FUNCTION "FC_LoadConfig" : Void
{ S7_Optimized_Access := 'TRUE' }
VERSION : 1.2
// =============================================================================
// Version_Recipe -- 00_Configuration.scl
// Central machine configuration -- called ONCE by OB100 (Startup) on every
// PLC power-up or program download.
//
// This file writes physical machine parameters (speed, limits, calibration, etc.)
// to DBs at PLC startup. Parameters that can be changed at runtime from HMI
// are NOT written here -- they remain as the DB initial values and revert to
// their initial values on warm-restart (NON_RETAIN DB).
//
// â”€â”€â”€ WHERE TO LOOK â”€â”€â”€â”€â”€â”€â”€â”€â”€â”€â”€â”€â”€â”€â”€â”€â”€â”€â”€â”€â”€â”€â”€â”€â”€â”€â”€â”€â”€â”€â”€â”€â”€â”€â”€â”€â”€â”€â”€â”€â”€â”€â”€â”€â”€â”€â”€â”€â”€â”€â”€â”€â”€â”€â”€â”€â”€â”€â”€
//   Maximum axis velocity        â†’ Section 1: MaxVelocity, RapidVelocity
//   Homing speed and mode        â†’ Section 2: HomeVelocity, HomingMode
//   Tool slot and angle settings â†’ Section 3: ToolCount, AutoCalcAngles
//   Spindle min/max RPM          â†’ Section 4: MinSpeed, MaxSpeed
//   Jog speed and step size      â†’ Section 5: JogSpeed, JogIncrement
//   Linear ruler stroke          â†’ Section 6: Phys_Max
//   Cylinder config reference    â†’ Section 7: see 02_DataBlocks.scl DB_Cylinder1
//   HMI initial values           â†’ Section 8: FeedrateOverride, ProductSelect
//   Test/commissioning bypass    â†’ Section 9: Bypass_EStop, Bypass_Door...
//   All timer PT values          â†’ Section 10: cylinder waits + process timeouts
//
// â”€â”€â”€ HMI SCREEN MAP â”€â”€â”€â”€â”€â”€â”€â”€â”€â”€â”€â”€â”€â”€â”€â”€â”€â”€â”€â”€â”€â”€â”€â”€â”€â”€â”€â”€â”€â”€â”€â”€â”€â”€â”€â”€â”€â”€â”€â”€â”€â”€â”€â”€â”€â”€â”€â”€â”€â”€â”€â”€â”€â”€â”€â”€â”€â”€
// Lists which tags are used on which HMI screen.
// "(â†’PLC)" = HMI writes, PLC reads  |  "(PLCâ†’)" = PLC writes, HMI reads (read-only)
//
// â”Œâ”€ MAIN SCREEN / STATUS LAMPS â”€â”€â”€â”€â”€â”€â”€â”€â”€â”€â”€â”€â”€â”€â”€â”€â”€â”€â”€â”€â”€â”€â”€â”€â”€â”€â”€â”€â”€â”€â”€â”€â”€â”€â”€â”€â”€â”€â”€â”€â”€â”€â”€â”€â”
// â”‚  DB_HMI.StatusMsg          (String[50])  PLCâ†’  "Running/Stopped/Errorâ€¦"â”‚
// â”‚  DB_HMI.IsRunning          (Bool)        PLCâ†’  Green lamp               â”‚
// â”‚  DB_HMI.IsPaused           (Bool)        PLCâ†’  Yellow lamp              â”‚
// â”‚  DB_HMI.HasError           (Bool)        PLCâ†’  Red lamp                 â”‚
// â”‚  DB_HMI.ActualX            (Real, mm)    PLCâ†’  X axis current position  â”‚
// â”‚  DB_HMI.ActualZ            (Real, mm)    PLCâ†’  Z axis current position  â”‚
// â”‚  DB_HMI.CurrentLine        (Int)         PLCâ†’  Active recipe line       â”‚
// â”‚  DB_HMI.ProgressPercent    (Real, %)     PLCâ†’  Progress bar             â”‚
// â”‚  DB_HMI.ElapsedSeconds     (DInt, s)     PLCâ†’  Cycle elapsed time       â”‚
// â”‚  DB_HMI.CycleCount         (Int)         PLCâ†’  Completed cycle count    â”‚
// â””â”€â”€â”€â”€â”€â”€â”€â”€â”€â”€â”€â”€â”€â”€â”€â”€â”€â”€â”€â”€â”€â”€â”€â”€â”€â”€â”€â”€â”€â”€â”€â”€â”€â”€â”€â”€â”€â”€â”€â”€â”€â”€â”€â”€â”€â”€â”€â”€â”€â”€â”€â”€â”€â”€â”€â”€â”€â”€â”€â”€â”€â”€â”€â”€â”€â”€â”€â”€â”€â”€â”€â”€â”€â”€â”˜
//
// â”Œâ”€ MAIN SCREEN / BUTTONS â”€â”€â”€â”€â”€â”€â”€â”€â”€â”€â”€â”€â”€â”€â”€â”€â”€â”€â”€â”€â”€â”€â”€â”€â”€â”€â”€â”€â”€â”€â”€â”€â”€â”€â”€â”€â”€â”€â”€â”€â”€â”€â”€â”€â”€â”€â”€â”€â”€â”€â”
// â”‚  DB_HMI.Btn_Start          (Bool)        â†’PLC  Start (rising edge)      â”‚
// â”‚  DB_HMI.Btn_Stop           (Bool)        â†’PLC  Stop (controlled stop)   â”‚
// â”‚  DB_HMI.Btn_Pause          (Bool)        â†’PLC  Pause                    â”‚
// â”‚  DB_HMI.Btn_Continue       (Bool)        â†’PLC  Resume from pause        â”‚
// â”‚  DB_HMI.Btn_AckError       (Bool)        â†’PLC  Acknowledge error + STOP â”‚
// â”‚  DB_HMI.Btn_Reset          (Bool)        â†’PLC  Full reset + STOPPED     â”‚
// â”‚  DB_HMI.ProductSelect      (Int, 1-5)    â†’PLC  Which program to run     â”‚
// â”‚  DB_HMI.FeedrateOverride   (Real, %)     â†’PLC  G1 speed multiplier      â”‚
// â”‚  DB_HMI.RapidOverride      (Real, %)     â†’PLC  G0 speed multiplier      â”‚
// â”‚  DB_HMI.SingleStepMode     (Bool)        â†’PLC  Line-by-line execution   â”‚
// â””â”€â”€â”€â”€â”€â”€â”€â”€â”€â”€â”€â”€â”€â”€â”€â”€â”€â”€â”€â”€â”€â”€â”€â”€â”€â”€â”€â”€â”€â”€â”€â”€â”€â”€â”€â”€â”€â”€â”€â”€â”€â”€â”€â”€â”€â”€â”€â”€â”€â”€â”€â”€â”€â”€â”€â”€â”€â”€â”€â”€â”€â”€â”€â”€â”€â”€â”€â”€â”€â”€â”€â”€â”€â”€â”˜
//
// â”Œâ”€ ERROR / ALARM SCREEN â”€â”€â”€â”€â”€â”€â”€â”€â”€â”€â”€â”€â”€â”€â”€â”€â”€â”€â”€â”€â”€â”€â”€â”€â”€â”€â”€â”€â”€â”€â”€â”€â”€â”€â”€â”€â”€â”€â”€â”€â”€â”€â”€â”€â”€â”€â”€â”€â”€â”€â”€â”
// â”‚  DB_Error.Active           (Bool)        PLCâ†’  Is there an active error? â”‚
// â”‚  DB_Error.Code             (Word, hex)   PLCâ†’  Error code (e.g. 0x0401) â”‚
// â”‚  DB_Error.Details          (String[80])  PLCâ†’  Error description text   â”‚
// â”‚  DB_Error.Severity         (Byte)        PLCâ†’  3=fatal, 2=error, 1=warn â”‚
// â”‚  DB_Error.Source           (String[20])  PLCâ†’  "Safety"/"Axis"/"Limit"  â”‚
// â”‚  DB_Error.TimeStamp        (DTL)         PLCâ†’  Error timestamp          â”‚
// â”‚  -- Alarm History (last 10) â”€â”€â”€â”€â”€â”€â”€â”€â”€â”€â”€â”€â”€â”€â”€â”€â”€â”€â”€â”€â”€â”€â”€â”€â”€â”€â”€â”€â”€â”€â”€â”€â”€â”€â”€â”€â”€â”€â”€â”€â”€â”€â”€â”€â”‚
// â”‚  DB_Error.History_Code[1..10]   (Word)   PLCâ†’  Last 10 error codes      â”‚
// â”‚  DB_Error.History_Details[1..10](String) PLCâ†’  Last 10 error details    â”‚
// â”‚  DB_Error.History_Time[1..10]   (DTL)    PLCâ†’  Last 10 error timestamps â”‚
// â””â”€â”€â”€â”€â”€â”€â”€â”€â”€â”€â”€â”€â”€â”€â”€â”€â”€â”€â”€â”€â”€â”€â”€â”€â”€â”€â”€â”€â”€â”€â”€â”€â”€â”€â”€â”€â”€â”€â”€â”€â”€â”€â”€â”€â”€â”€â”€â”€â”€â”€â”€â”€â”€â”€â”€â”€â”€â”€â”€â”€â”€â”€â”€â”€â”€â”€â”€â”€â”€â”€â”€â”€â”€â”€â”˜
//
// â”Œâ”€ MANUAL SCREEN / MOTION â”€â”€â”€â”€â”€â”€â”€â”€â”€â”€â”€â”€â”€â”€â”€â”€â”€â”€â”€â”€â”€â”€â”€â”€â”€â”€â”€â”€â”€â”€â”€â”€â”€â”€â”€â”€â”€â”€â”€â”€â”€â”€â”€â”€â”€â”€â”€â”€â”€â”
// â”‚  DB_Manual.ManualModeActive (Bool)       â†’PLC  Enable/disable manual modeâ”‚
// â”‚  DB_Manual.SelectedAxis    (Int, 0-3)    â†’PLC  0=X 1=Z 2=Tool 3=Spindle â”‚
// â”‚  DB_Manual.Btn_JogPlus     (Bool)        â†’PLC  Positive direction jog   â”‚
// â”‚  DB_Manual.Btn_JogMinus    (Bool)        â†’PLC  Negative direction jog   â”‚
// â”‚  DB_Manual.JogSpeed        (Real, mm/s)  â†’PLC  Jog speed                â”‚
// â”‚  DB_Manual.Btn_StepPlus    (Bool)        â†’PLC  +JogIncrement step       â”‚
// â”‚  DB_Manual.Btn_StepMinus   (Bool)        â†’PLC  -JogIncrement step       â”‚
// â”‚  DB_Manual.JogIncrement    (Real, mm)    â†’PLC  Step size                â”‚
// â”‚  DB_Manual.MoveToPosition  (Real, mm)    â†’PLC  Target absolute position â”‚
// â”‚  DB_Manual.Btn_MoveAbsolute(Bool)        â†’PLC  Start absolute move      â”‚
// â”‚  DB_Manual.Btn_HomeAll     (Bool)        â†’PLC  Home all axes             â”‚
// â”‚  DB_Manual.Btn_GoSafe      (Bool)        â†’PLC  Move to safe position    â”‚
// â”‚  DB_Manual.Btn_GoZero      (Bool)        â†’PLC  Move to zero position    â”‚
// â”‚  DB_Manual.SelectedAxisPos (Real, mm)    PLCâ†’  Selected axis position   â”‚
// â”‚  DB_Manual.SelectedAxisName(String)      PLCâ†’  "X" / "Z" / "Tool"      â”‚
// â”‚  DB_Manual.JogBusy         (Bool)        PLCâ†’  Motion in progress       â”‚
// â””â”€â”€â”€â”€â”€â”€â”€â”€â”€â”€â”€â”€â”€â”€â”€â”€â”€â”€â”€â”€â”€â”€â”€â”€â”€â”€â”€â”€â”€â”€â”€â”€â”€â”€â”€â”€â”€â”€â”€â”€â”€â”€â”€â”€â”€â”€â”€â”€â”€â”€â”€â”€â”€â”€â”€â”€â”€â”€â”€â”€â”€â”€â”€â”€â”€â”€â”€â”€â”€â”€â”€â”€â”€â”€â”˜
//
// â”Œâ”€ MANUAL SCREEN / SPINDLE â”€â”€â”€â”€â”€â”€â”€â”€â”€â”€â”€â”€â”€â”€â”€â”€â”€â”€â”€â”€â”€â”€â”€â”€â”€â”€â”€â”€â”€â”€â”€â”€â”€â”€â”€â”€â”€â”€â”€â”€â”€â”€â”€â”€â”€â”€â”€â”€â”
// â”‚  DB_Manual.Btn_SpindleStart(Bool)        â†’PLC  Start spindle            â”‚
// â”‚  DB_Manual.Btn_SpindleStop (Bool)        â†’PLC  Stop spindle             â”‚
// â”‚  DB_Manual.Manual_SpindleSpeed (Real,RPM)â†’PLC  Manual spindle speed     â”‚
// â”‚  DB_Manual.Manual_SpindleDir   (Int)     â†’PLC  1=CW, -1=CCW            â”‚
// â”‚  DB_Spindle.IsRunning      (Bool)        PLCâ†’  Spindle running          â”‚
// â”‚  DB_Spindle.AtSpeed        (Bool)        PLCâ†’  Speed stable             â”‚
// â”‚  DB_Spindle.ActualSpeed    (Real, RPM)   PLCâ†’  Current spindle speed    â”‚
// â””â”€â”€â”€â”€â”€â”€â”€â”€â”€â”€â”€â”€â”€â”€â”€â”€â”€â”€â”€â”€â”€â”€â”€â”€â”€â”€â”€â”€â”€â”€â”€â”€â”€â”€â”€â”€â”€â”€â”€â”€â”€â”€â”€â”€â”€â”€â”€â”€â”€â”€â”€â”€â”€â”€â”€â”€â”€â”€â”€â”€â”€â”€â”€â”€â”€â”€â”€â”€â”€â”€â”€â”€â”€â”€â”˜
//
// â”Œâ”€ MANUAL SCREEN / MANAGE (Drive Management) â”€â”€â”€â”€â”€â”€â”€â”€â”€â”€â”€â”€â”€â”€â”€â”€â”€â”€â”€â”€â”€â”€â”€â”€â”€â”€â”€â”€â”€â”
// â”‚  DB_HMI.Btn_Contactor_X    (Bool)        â†’PLC  X drive contactor        â”‚
// â”‚  DB_HMI.Btn_Contactor_Z    (Bool)        â†’PLC  Z drive contactor        â”‚
// â”‚  DB_HMI.Btn_Contactor_Tool (Bool)        â†’PLC  Tool drive contactor     â”‚
// â”‚  DB_HMI.Btn_Enable_X       (Bool)        â†’PLC  X drive enable signal    â”‚
// â”‚  DB_HMI.Btn_Enable_Z       (Bool)        â†’PLC  Z drive enable signal    â”‚
// â”‚  DB_HMI.Contactor_X_On     (Bool)        PLCâ†’  X contactor feedback     â”‚
// â”‚  DB_HMI.Contactor_Z_On     (Bool)        PLCâ†’  Z contactor feedback     â”‚
// â”‚  DB_HMI.Enable_X_On        (Bool)        PLCâ†’  X enable feedback        â”‚
// â”‚  NOTE: Contactor and Enable must be toggle buttons (maintained),         â”‚
// â”‚        NOT momentary.                                                    â”‚
// â””â”€â”€â”€â”€â”€â”€â”€â”€â”€â”€â”€â”€â”€â”€â”€â”€â”€â”€â”€â”€â”€â”€â”€â”€â”€â”€â”€â”€â”€â”€â”€â”€â”€â”€â”€â”€â”€â”€â”€â”€â”€â”€â”€â”€â”€â”€â”€â”€â”€â”€â”€â”€â”€â”€â”€â”€â”€â”€â”€â”€â”€â”€â”€â”€â”€â”€â”€â”€â”€â”€â”€â”€â”€â”€â”˜
//
// â”Œâ”€ TOOL PAGE â”€â”€â”€â”€â”€â”€â”€â”€â”€â”€â”€â”€â”€â”€â”€â”€â”€â”€â”€â”€â”€â”€â”€â”€â”€â”€â”€â”€â”€â”€â”€â”€â”€â”€â”€â”€â”€â”€â”€â”€â”€â”€â”€â”€â”€â”€â”€â”€â”€â”€â”€â”€â”€â”€â”€â”€â”€â”€â”€â”€â”€â”€â”
// â”‚  DB_MachineConfig.ToolCount         (Int, 1-4)  â†’PLC  Slot count        â”‚
// â”‚  DB_ToolConfig.AutoCalcAngles       (Bool)       â†’PLC  Auto angle calc  â”‚
// â”‚  DB_ToolConfig.ToolStepAngle_Calc   (Real, Â°)   PLCâ†’  Calculated step   â”‚
// â”‚  DB_ToolConfig.Tool1_Position       (Real, Â°)   PLCâ†’  Slot 1 angle      â”‚
// â”‚  DB_ToolConfig.Tool2_Position       (Real, Â°)   PLCâ†’  Slot 2 angle      â”‚
// â”‚  DB_ToolConfig.Tool3_Position       (Real, Â°)   PLCâ†’  Slot 3 angle      â”‚
// â”‚  DB_ToolConfig.Tool4_Position       (Real, Â°)   PLCâ†’  Slot 4 angle      â”‚
// â”‚  DB_HMI.ToolSlotCode[1..4]          (Int)        â†’PLC  Slot code input  â”‚
// â”‚  DB_HMI.Btn_ApplyToolConfig         (Bool)       â†’PLC  Apply code       â”‚
// â”‚  DB_ToolConfig.ToolCode_List[1..4]  (Int)        PLCâ†’  Active slot code â”‚
// â”‚  NOTE: While AutoCalcAngles=TRUE, tool angles cannot be changed from     â”‚
// â”‚        HMI -- they are overwritten every scan. Set FALSE for manual anglesâ”‚
// â””â”€â”€â”€â”€â”€â”€â”€â”€â”€â”€â”€â”€â”€â”€â”€â”€â”€â”€â”€â”€â”€â”€â”€â”€â”€â”€â”€â”€â”€â”€â”€â”€â”€â”€â”€â”€â”€â”€â”€â”€â”€â”€â”€â”€â”€â”€â”€â”€â”€â”€â”€â”€â”€â”€â”€â”€â”€â”€â”€â”€â”€â”€â”€â”€â”€â”€â”€â”€â”€â”€â”€â”€â”€â”€â”˜
//
// â”Œâ”€ CYLINDER PAGE â”€â”€â”€â”€â”€â”€â”€â”€â”€â”€â”€â”€â”€â”€â”€â”€â”€â”€â”€â”€â”€â”€â”€â”€â”€â”€â”€â”€â”€â”€â”€â”€â”€â”€â”€â”€â”€â”€â”€â”€â”€â”€â”€â”€â”€â”€â”€â”€â”€â”€â”€â”€â”€â”€â”€â”€â”€â”€â”
// â”‚  DB_Cylinder1.ValveType    (Byte)        â†’PLC  1=5/2  2=5/3_blocked     â”‚
// â”‚  DB_Cylinder1.Cmd_Extend   (Bool)        â†’PLC  Extend: move to setpoint â”‚
// â”‚  DB_Cylinder1.Cmd_ExtendFull(Bool)       â†’PLC  Extend: full stroke      â”‚
// â”‚  DB_Cylinder1.Cmd_Retract  (Bool)        â†’PLC  Retract                  â”‚
// â”‚  DB_Cylinder1.Timeout_Extend(Time)       â†’PLC  Extend timeout (T#5S)    â”‚
// â”‚  DB_Cylinder1.Timeout_Retract(Time)      â†’PLC  Retract timeout (T#5S)   â”‚
// â”‚  DB_Cylinder1.State        (Int)         PLCâ†’  -1=EStop 0=Idle          â”‚
// â”‚                                                  1=Extending 2=Retractingâ”‚
// â”‚                                                  3=AtSetpoint 4=AtRetractâ”‚
// â”‚                                                 10=ERROR                 â”‚
// â”‚  DB_Cylinder1.StateText    (String[14])  PLCâ†’  State text               â”‚
// â”‚  DB_Cylinder1.AtSetpoint   (Bool)        PLCâ†’  Locked at setpoint       â”‚
// â”‚  DB_Cylinder1.AtRetract    (Bool)        PLCâ†’  At retract end           â”‚
// â”‚  DB_Cylinder1.Error        (Bool)        PLCâ†’  Active error             â”‚
// â”‚  DB_Cylinder1.ErrorID      (Word)        PLCâ†’  0x0501/0502/0503         â”‚
// â”‚  DB_LinearRuler1.Value      (Real, mm)    PLCâ†’  Ruler position           â”‚
// â”‚  DB_LinearRuler1.Valid       (Bool)        PLCâ†’  Sensor healthy?         â”‚
// â”‚  NOTE: Cmd_Extend AND Cmd_Retract TRUE simultaneously â†’ Hold (conflict  â”‚
// â”‚        protection). Purchase BLOCKED CENTER valve -- cylinder is          â”‚
// â”‚        mechanically locked in hold. Do NOT use EXHAUST CENTER.          â”‚
// â””â”€â”€â”€â”€â”€â”€â”€â”€â”€â”€â”€â”€â”€â”€â”€â”€â”€â”€â”€â”€â”€â”€â”€â”€â”€â”€â”€â”€â”€â”€â”€â”€â”€â”€â”€â”€â”€â”€â”€â”€â”€â”€â”€â”€â”€â”€â”€â”€â”€â”€â”€â”€â”€â”€â”€â”€â”€â”€â”€â”€â”€â”€â”€â”€â”€â”€â”€â”€â”€â”€â”€â”€â”€â”€â”˜
//
// â”Œâ”€ RULER CALIBRATION (Setup Screen) â”€â”€â”€â”€â”€â”€â”€â”€â”€â”€â”€â”€â”€â”€â”€â”€â”€â”€â”€â”€â”€â”€â”€â”€â”€â”€â”€â”€â”€â”€â”€â”€â”€â”€â”€â”€â”€â”€â”
// â”‚  DB_LinearRuler1.Raw_Min      (Int)       â†’PLC  AI raw min value         â”‚
// â”‚  DB_LinearRuler1.Raw_Max      (Int)       â†’PLC  AI raw max value         â”‚
// â”‚  DB_LinearRuler1.Phys_Min     (Real, mm)  â†’PLC  Physical ref at Raw_Min  â”‚
// â”‚  DB_LinearRuler1.Phys_Max     (Real, mm)  â†’PLC  Physical ref at Raw_Max  â”‚
// â”‚  DB_LinearRuler1.InvertSignal (Bool)      â†’PLC  TRUE=0Vâ†’high physical    â”‚
// â”‚  DB_LinearRuler1.Value        (Real, mm)  PLCâ†’  Scaled position (mm)     â”‚
// â”‚  DB_LinearRuler1.Valid        (Bool)      PLCâ†’  Sensor within range?     â”‚
// â”‚  NOTE: S7-1200 standard AI: 0V=0, 10V=27648 (4-20mA: 4mA=5530,20mA=27648â”‚
// â””â”€â”€â”€â”€â”€â”€â”€â”€â”€â”€â”€â”€â”€â”€â”€â”€â”€â”€â”€â”€â”€â”€â”€â”€â”€â”€â”€â”€â”€â”€â”€â”€â”€â”€â”€â”€â”€â”€â”€â”€â”€â”€â”€â”€â”€â”€â”€â”€â”€â”€â”€â”€â”€â”€â”€â”€â”€â”€â”€â”€â”€â”€â”€â”€â”€â”€â”€â”€â”€â”€â”€â”€â”€â”€â”˜
//
// â”Œâ”€ MACHINE LIMITS (Setup Screen) â”€â”€â”€â”€â”€â”€â”€â”€â”€â”€â”€â”€â”€â”€â”€â”€â”€â”€â”€â”€â”€â”€â”€â”€â”€â”€â”€â”€â”€â”€â”€â”€â”€â”€â”€â”€â”€â”€â”€â”€â”€â”
// â”‚  DB_MachineConfig.SoftLimit_MinX  (Real, mm)  â†’PLC  X software min      â”‚
// â”‚  DB_MachineConfig.SoftLimit_MaxX  (Real, mm)  â†’PLC  X software max      â”‚
// â”‚  DB_MachineConfig.SoftLimit_MinZ  (Real, mm)  â†’PLC  Z software min      â”‚
// â”‚  DB_MachineConfig.SoftLimit_MaxZ  (Real, mm)  â†’PLC  Z software max      â”‚
// â”‚  DB_MachineConfig.HomeVelocity    (Real, mm/s)â†’PLC  Homing speed        â”‚
// â”‚  DB_MachineConfig.SafePos_X/Z     (Real, mm)  â†’PLC  "Go Safe" target    â”‚
// â”‚  NOTE: These values are not written by FC_LoadConfig. Use DB initial     â”‚
// â”‚        values or change from HMI. Reverts to DB initial on PLC restart. â”‚
// â””â”€â”€â”€â”€â”€â”€â”€â”€â”€â”€â”€â”€â”€â”€â”€â”€â”€â”€â”€â”€â”€â”€â”€â”€â”€â”€â”€â”€â”€â”€â”€â”€â”€â”€â”€â”€â”€â”€â”€â”€â”€â”€â”€â”€â”€â”€â”€â”€â”€â”€â”€â”€â”€â”€â”€â”€â”€â”€â”€â”€â”€â”€â”€â”€â”€â”€â”€â”€â”€â”€â”€â”€â”€â”€â”˜
//
// â”Œâ”€ PRODUCTION COUNTERS â”€â”€â”€â”€â”€â”€â”€â”€â”€â”€â”€â”€â”€â”€â”€â”€â”€â”€â”€â”€â”€â”€â”€â”€â”€â”€â”€â”€â”€â”€â”€â”€â”€â”€â”€â”€â”€â”€â”€â”€â”€â”€â”€â”€â”€â”€â”€â”€â”€â”€â”€â”€â”
// â”‚  DB_Production.TotalOK     (DInt)        PLCâ†’  Successful cycle count   â”‚
// â”‚  DB_Production.TotalNOK    (DInt)        PLCâ†’  Failed cycle count       â”‚
// â”‚  DB_Production.TotalStopped(DInt)        PLCâ†’  Operator stop count      â”‚
// â”‚  DB_Production.LastResult  (Byte)        PLCâ†’  1=OK, 2=NOK, 3=STOP      â”‚
// â”‚  DB_Production.LastErrorCode(Word)       PLCâ†’  Last error code          â”‚
// â”‚  DB_HMI.Btn_ProdReset      (Bool)        â†’PLC  Reset counters           â”‚
// â””â”€â”€â”€â”€â”€â”€â”€â”€â”€â”€â”€â”€â”€â”€â”€â”€â”€â”€â”€â”€â”€â”€â”€â”€â”€â”€â”€â”€â”€â”€â”€â”€â”€â”€â”€â”€â”€â”€â”€â”€â”€â”€â”€â”€â”€â”€â”€â”€â”€â”€â”€â”€â”€â”€â”€â”€â”€â”€â”€â”€â”€â”€â”€â”€â”€â”€â”€â”€â”€â”€â”€â”€â”€â”€â”˜
//
// â”Œâ”€ BYPASS / TEST MODE â”€â”€â”€â”€â”€â”€â”€â”€â”€â”€â”€â”€â”€â”€â”€â”€â”€â”€â”€â”€â”€â”€â”€â”€â”€â”€â”€â”€â”€â”€â”€â”€â”€â”€â”€â”€â”€â”€â”€â”€â”€â”€â”€â”€â”€â”€â”€â”€â”€â”€â”€â”€â”€â”
// â”‚  DB_HMI.Bypass_EStop       (Bool)        â†’PLC  âš ï¸ TEST ONLY             â”‚
// â”‚  DB_HMI.Bypass_Door        (Bool)        â†’PLC  âš ï¸ TEST ONLY             â”‚
// â”‚  DB_HMI.Bypass_AirPressure (Bool)        â†’PLC  âš ï¸ TEST ONLY             â”‚
// â”‚  DB_HMI.Bypass_Drives      (Bool)        â†’PLC  âš ï¸ TEST ONLY             â”‚
// â”‚  âš ï¸ The PLC does NOT clear bypasses while active. The operator must      â”‚
// â”‚     turn them off manually. Verify before going into production.         â”‚
// â”‚  NOTE: DB_HMI.Bypass_Spindle and Bypass_ToolChanger are defined but     â”‚
// â”‚        not used in the safety monitor -- do not connect them.            â”‚
// â””â”€â”€â”€â”€â”€â”€â”€â”€â”€â”€â”€â”€â”€â”€â”€â”€â”€â”€â”€â”€â”€â”€â”€â”€â”€â”€â”€â”€â”€â”€â”€â”€â”€â”€â”€â”€â”€â”€â”€â”€â”€â”€â”€â”€â”€â”€â”€â”€â”€â”€â”€â”€â”€â”€â”€â”€â”€â”€â”€â”€â”€â”€â”€â”€â”€â”€â”€â”€â”€â”€â”€â”€â”€â”€â”˜
// =============================================================================
// -----------------------------------------------------------------------------
// FC_LoadConfig -- Runs once at PLC startup (called by OB100)
// Values here can be thought of as the PLC "factory defaults".
// Parameters that can be changed at runtime from HMI are NOT written here --
// the initial value in the DB definition applies.
// -----------------------------------------------------------------------------

BEGIN


	// =========================================================================
	// SECTION 1 -- AXIS VELOCITY LIMITS (mm/s)
	// â”€â”€â”€â”€â”€â”€â”€â”€â”€â”€â”€â”€â”€â”€â”€â”€â”€â”€â”€â”€â”€â”€â”€â”€â”€â”€â”€â”€â”€â”€â”€â”€â”€â”€â”€â”€â”€â”€â”€â”€â”€â”€â”€â”€â”€â”€â”€â”€â”€â”€â”€â”€â”€â”€â”€â”€â”€â”€â”€â”€â”€â”€â”€â”€â”€â”€â”€â”€â”€â”€â”€â”€â”€
	// âš ï¸ These values MUST match the Technology Object (TO) settings in TIA Portal.
	//    If the TO has a different limit, the PLC may report an error.
	//    Should not be changed from HMI -- edit here instead.
	// â”€â”€â”€â”€â”€â”€â”€â”€â”€â”€â”€â”€â”€â”€â”€â”€â”€â”€â”€â”€â”€â”€â”€â”€â”€â”€â”€â”€â”€â”€â”€â”€â”€â”€â”€â”€â”€â”€â”€â”€â”€â”€â”€â”€â”€â”€â”€â”€â”€â”€â”€â”€â”€â”€â”€â”€â”€â”€â”€â”€â”€â”€â”€â”€â”€â”€â”€â”€â”€â”€â”€â”€â”€
	//  MaxVelocity   : Must match "Maximum velocity" in TO
	//  RapidVelocity : Used for G0 command (in recipe)
	//  MinVelocity   : Must match "Minimum velocity" in TO
	// =========================================================================
	"DB_MachineConfig".MaxVelocity := 40.0;   // mm/s -- match TO max velocity
	"DB_MachineConfig".RapidVelocity := 30.0;   // mm/s -- G0 (rapid move) speed
	"DB_MachineConfig".MinVelocity := 0.001;    // mm/s -- match TO min velocity
	"DB_MachineConfig".FeedrateConvFactor := 60.0;    // divisor: recipe F (mm/min) / this = axis velocity (mm/s)
	// Standard mm/minâ†’mm/s = divide by 60; adjust if TO uses different units

	// =========================================================================
	// SECTION 2 -- HOMING (REFERENCE SEEK)
	// â”€â”€â”€â”€â”€â”€â”€â”€â”€â”€â”€â”€â”€â”€â”€â”€â”€â”€â”€â”€â”€â”€â”€â”€â”€â”€â”€â”€â”€â”€â”€â”€â”€â”€â”€â”€â”€â”€â”€â”€â”€â”€â”€â”€â”€â”€â”€â”€â”€â”€â”€â”€â”€â”€â”€â”€â”€â”€â”€â”€â”€â”€â”€â”€â”€â”€â”€â”€â”€â”€â”€â”€â”€
	//  HomingMode:
	//    0 = Passive  â†’ Motor does not move, encoder is zeroed at current position
	//    2 = Active   â†’ Moves to reference switch, encoder is zeroed
	//    3 = Active+Zero â†’ Moves to reference switch, set to HomeOffset_X/Z value
	//                    (recommended mode for production)
	//
	//  HomeVelocity and HomeOffset_X/Z are defined as initial values in
	//  DB_MachineConfig and can be edited from the HMI Machine Limits screen.
	//  Writing here will always reset to the same value on restart.
	// =========================================================================
	"DB_Manual".HomingMode := 3;   // 0=Passive | 2=Active | 3=Active+Zero (recommended)
	"DB_MachineConfig".PostHome_Clearance := 0.0;  // mm -- clearance distance from PNP zone after homing
	"DB_MachineConfig".HomeVelocity := 5.0;         // mm/s -- speed for pre/post-homing clearance move
	// NOTE: MC_Home search speed comes from TO, PLC cannot change it
	"DB_MachineConfig".AlwaysHomeOnAutoStart := TRUE; // Home all axes on every auto start (set FALSE for fast test cycles)

	// =========================================================================
	// SECTION 3 -- TOOL CHANGER
	// â”€â”€â”€â”€â”€â”€â”€â”€â”€â”€â”€â”€â”€â”€â”€â”€â”€â”€â”€â”€â”€â”€â”€â”€â”€â”€â”€â”€â”€â”€â”€â”€â”€â”€â”€â”€â”€â”€â”€â”€â”€â”€â”€â”€â”€â”€â”€â”€â”€â”€â”€â”€â”€â”€â”€â”€â”€â”€â”€â”€â”€â”€â”€â”€â”€â”€â”€â”€â”€â”€â”€â”€â”€
	//  ToolCount: How many slots are physically installed (1-4)
	//    â†’ FC_ToolAngleCalc automatically calculates angles based on this value
	//    â†’ Can also be changed on the HMI Tool page (runtime)
	//
	//  AutoCalcAngles = TRUE  â†’ Equally spaced angles based on ToolCount
	//                           (2 slots: 0Â°/180Â°, 3 slots: 0Â°/120Â°/240Â°, etc.)
	//  AutoCalcAngles = FALSE â†’ Tool1..4_Position can be entered manually from HMI
	//                           (use when unequal angles are needed)
	//
	//  CurrentTool: Which slot is active at startup (usually 1)
	// =========================================================================
	"DB_MachineConfig".ToolCount := 3;     // Physical slot count
	"DB_ToolConfig".AutoCalcAngles := TRUE;  // Automatic angle calculation
	"DB_ToolConfig".CurrentTool := 1;     // Initial active slot

	// =========================================================================
	// SECTION 4 -- SPINDLE SPEED
	// â”€â”€â”€â”€â”€â”€â”€â”€â”€â”€â”€â”€â”€â”€â”€â”€â”€â”€â”€â”€â”€â”€â”€â”€â”€â”€â”€â”€â”€â”€â”€â”€â”€â”€â”€â”€â”€â”€â”€â”€â”€â”€â”€â”€â”€â”€â”€â”€â”€â”€â”€â”€â”€â”€â”€â”€â”€â”€â”€â”€â”€â”€â”€â”€â”€â”€â”€â”€â”€â”€â”€â”€â”€
	//  MinSpeed      : Commands below this value are clamped to this value
	//  MaxSpeed      : Commands above this value are clamped to this value
	//  DefaultSpeed  : Default speed in manual mode (initial Manual_SpindleSpeed)
	//  SpeedTolerance: Tolerance for "AtSpeed" decision -- keep small (Â±5% recommended)
	//  SpeedOverride : 100% = normal, can be changed at runtime from HMI
	//
	//  âš ï¸ MaxSpeed must not exceed motor or coupling component ratings
	// =========================================================================
	"DB_Spindle".MinSpeed := 100.0;   // RPM -- lower limit
	"DB_Spindle".MaxSpeed := 3000.0;  // RPM -- upper limit (do not exceed motor max)
	"DB_Spindle".DefaultSpeed := 1000.0;  // RPM -- manual mode initial value
	"DB_Spindle".SpeedTolerance := 5.0;     // % -- AtSpeed tolerance
	"DB_Spindle".SpeedOverride := 100.0;   // % -- 100% at startup (normal)
	"DB_MachineConfig".SpindleMaxRPM := 2400.0;  // RPM -- denominator for proportional MandrelLock wait (ITEM-28)
	"DB_MachineConfig".SpindleStopSafeTime := T#10S;   // Full-speed decel safety margin -- tune to measured VFD ramp + margin

	// =========================================================================
	// SECTION 5 -- MANUAL MODE DEFAULTS
	// â”€â”€â”€â”€â”€â”€â”€â”€â”€â”€â”€â”€â”€â”€â”€â”€â”€â”€â”€â”€â”€â”€â”€â”€â”€â”€â”€â”€â”€â”€â”€â”€â”€â”€â”€â”€â”€â”€â”€â”€â”€â”€â”€â”€â”€â”€â”€â”€â”€â”€â”€â”€â”€â”€â”€â”€â”€â”€â”€â”€â”€â”€â”€â”€â”€â”€â”€â”€â”€â”€â”€â”€â”€
	//  JogSpeed      : Speed used when jog button is pressed
	//                  Can be connected to a slider/input field on HMI Manual screen
	//  JogIncrement  : Distance traveled per press on "Step" button
	//  ToolStepAngle : Rotation angle for CW/CCW buttons on Manual Tool screen
	//                  (e.g. 90Â° can be used to step slot-to-slot)
	//  Manual_SpindleSpeed: Initial speed on manual spindle screen
	//  Manual_SpindleDir  : 1=CW (clockwise), -1=CCW (counter-clockwise)
	// =========================================================================
	"DB_Manual".JogSpeed := 30.0;   // mm/s
	"DB_Manual".JogIncrement := 1.0;    // mm -- step size
	"DB_Manual".ToolStepAngle := 120.0;   // degrees -- tool step angle
	"DB_Manual".Manual_SpindleSpeed := 500.0;  // RPM
	"DB_Manual".Manual_SpindleDir := 1;      // 1=CW | -1=CCW

	// =========================================================================
	// SECTION 6 -- LINEAR RULER CALIBRATION
	// â”€â”€â”€â”€â”€â”€â”€â”€â”€â”€â”€â”€â”€â”€â”€â”€â”€â”€â”€â”€â”€â”€â”€â”€â”€â”€â”€â”€â”€â”€â”€â”€â”€â”€â”€â”€â”€â”€â”€â”€â”€â”€â”€â”€â”€â”€â”€â”€â”€â”€â”€â”€â”€â”€â”€â”€â”€â”€â”€â”€â”€â”€â”€â”€â”€â”€â”€â”€â”€â”€â”€â”€â”€
	//  S7-1200 AI module standard output values:
	//    0 V  (or 4  mA) â†’ Raw_Min  (typically 0 or 5530)
	//    10 V (or 20 mA) â†’ Raw_Max  (typically 27648)
	//
	//  Phys_Min / Phys_Max: Mechanical stroke limits of the sensor (mm)
	//    Example: For a ruler with 0-200 mm stroke: Phys_Min=0, Phys_Max=200
	//
	//  âš ï¸ Always update Phys_Max according to the sensor stroke.
	//  These values revert here on restart -- for permanent changes write here,
	//  changes made only from HMI will be lost on restart.
	// =========================================================================
	"DB_Cylinder_LinearRuler_BackSupport".Raw_Min := 0;       // AI at full extend (~0V)
	"DB_Cylinder_LinearRuler_BackSupport".Raw_Max := 31433;   // AI at full retract (measured; update once hardware is within 0-10V)
	"DB_Cylinder_LinearRuler_BackSupport".Phys_Min := 0.0;     // mm physical reference at Raw_Min end
	"DB_Cylinder_LinearRuler_BackSupport".Phys_Max := 300.0;   // mm physical reference at Raw_Max end (full stroke)
	"DB_Cylinder_LinearRuler_BackSupport".InvertSignal := TRUE;    // Sensor wired reverse: 0V = full extend (300mm), ~10V = retracted (0mm)

	// â”€â”€ CMD=40 gain defaults â”€â”€â”€â”€â”€â”€â”€â”€â”€â”€â”€â”€â”€â”€â”€â”€â”€â”€â”€â”€â”€â”€â”€â”€â”€â”€â”€â”€â”€â”€â”€â”€â”€â”€â”€â”€â”€â”€â”€â”€â”€â”€â”€â”€â”€â”€â”€â”€â”€â”€
	// TargetPos = Param Ã— Cmd40_Gain (mm). Default 10.0 (no scaling).
	// Tune on-site: measure how far BackSupport travels per Param unit and update.
	// Example: if Param=20 should send BackSupport to 200mm â†’ Cmd40_Gain = 10.0
	"DB_Cylinder_BackSupport".Cmd40_Gain := 10.0;   // BackSupport: mm per CMD=40 Param unit

	// =========================================================================
	// SECTION 7 -- PNEUMATIC CYLINDER CONFIGURATION REFERENCE
	// â”€â”€â”€â”€â”€â”€â”€â”€â”€â”€â”€â”€â”€â”€â”€â”€â”€â”€â”€â”€â”€â”€â”€â”€â”€â”€â”€â”€â”€â”€â”€â”€â”€â”€â”€â”€â”€â”€â”€â”€â”€â”€â”€â”€â”€â”€â”€â”€â”€â”€â”€â”€â”€â”€â”€â”€â”€â”€â”€â”€â”€â”€â”€â”€â”€â”€â”€â”€â”€â”€â”€â”€â”€
	//  Cylinder parameters (ValveType, MaxPos, TargetPos, Timeout, UseRulerPos)
	//  are VAR_INPUT in FB_CylinderControl. In optimized S7 blocks VAR_INPUT
	//  fields cannot be written from an FC at runtime. Factory defaults must be
	//  set in the BEGIN section of DB_Cylinder1 in 02_DataBlocks.scl.
	//
	//  Current Cylinder 1 factory defaults (02_DataBlocks.scl â†’ DB_Cylinder1):
	//    ValveType       = 3       (5/3 blocked center -- piston locked in hold)
	//    UseRulerPos     = TRUE    (analog position control via DB_LinearRuler)
	//    TargetPos       = 300.0   (mm -- default: full extend)
	//    MaxPos          = 300.0   (mm -- software extend clamp)
	//    ExtendOffset    = 5.0     (mm -- tune on site)
	//    RetractOffset   = 5.0     (mm -- tune on site)
	//    Tolerance       = 2.0     (mm -- AtTarget window)
	//    Timeout_Extend  = T#5S
	//    Timeout_Retract = T#5S
	//
	//  âš ï¸ VALVE TYPE SELECTION IS CRITICAL:
	//    ValveType=2 BLOCKED CENTER â†’ Piston mechanically locked in hold. âœ… USE THIS
	//    ValveType=3 EXHAUST CENTER â†’ Piston free to move in hold.        âŒ Do not use
	// =========================================================================
	// (No runtime writes here -- edit 02_DataBlocks.scl DB_Cylinder1 BEGIN section)

	// =========================================================================
	// SECTION 8 -- HMI INITIAL VALUES
	// â”€â”€â”€â”€â”€â”€â”€â”€â”€â”€â”€â”€â”€â”€â”€â”€â”€â”€â”€â”€â”€â”€â”€â”€â”€â”€â”€â”€â”€â”€â”€â”€â”€â”€â”€â”€â”€â”€â”€â”€â”€â”€â”€â”€â”€â”€â”€â”€â”€â”€â”€â”€â”€â”€â”€â”€â”€â”€â”€â”€â”€â”€â”€â”€â”€â”€â”€â”€â”€â”€â”€â”€â”€
	//  FeedrateOverride: Speed multiplier for recipe G1 moves.
	//    100% = normal speed, 50% = half speed, 200% = double speed
	//    HMI slider should be connected to this tag (recommend min 50, max 200)
	//  RapidOverride: Same logic for G0 rapid moves
	//  ProductSelect: Which program is active at startup (1-5)
	// =========================================================================
	"DB_HMI".FeedrateOverride := 100.0;   // % -- initial feed rate multiplier
	"DB_HMI".RapidOverride := 100.0;   // % -- initial rapid rate multiplier
	"DB_HMI".SingleStepMode := FALSE;   // Line-by-line mode off
	"DB_HMI".ProductSelect := 1;       // Initial program selection

	// =========================================================================
	// SECTION 9 -- SAFETY BYPASSES
	// â”€â”€â”€â”€â”€â”€â”€â”€â”€â”€â”€â”€â”€â”€â”€â”€â”€â”€â”€â”€â”€â”€â”€â”€â”€â”€â”€â”€â”€â”€â”€â”€â”€â”€â”€â”€â”€â”€â”€â”€â”€â”€â”€â”€â”€â”€â”€â”€â”€â”€â”€â”€â”€â”€â”€â”€â”€â”€â”€â”€â”€â”€â”€â”€â”€â”€â”€â”€â”€â”€â”€â”€â”€
	//  âš ï¸âš ï¸ WARNING: These bypasses are for commissioning and testing only!
	//  Verify that ALL are FALSE before production.
	//
	//  PLC resets these to FALSE on every restart (safe default).
	//  Show a warning on HMI when any bypass is active (AnyBypassActive tag recommended).
	//
	//  Bypass_EStop       : Ignore physical E-Stop circuit
	//  Bypass_Door        : Ignore safety door sensor
	//  Bypass_AirPressure : Ignore air pressure sensor
	//  Bypass_Drives      : Ignore drive ready signal
	//
	//  Bypass_ToolAxis    : This bypass is DIFFERENT -- set TRUE if the tool axis
	//    (turret) is NOT physically connected to this machine.
	//    This is a hardware presence flag, not a safety bypass.
	//
	//  âš ï¸ NOTE: DB_HMI.Bypass_Spindle and DB_HMI.Bypass_ToolChanger are defined
	//    but not used in the safety monitor. Do not connect them to HMI.
	// =========================================================================
	"DB_HMI".Bypass_EStop := FALSE;
	"DB_HMI".Bypass_Door := TRUE; // NOT USED -- reserved for future use
	"DB_HMI".Bypass_AirPressure := TRUE; // NOT USED -- reserved for future use
	"DB_HMI".Bypass_Drives := FALSE;
	"DB_HMI".Bypass_Spindle := FALSE;
	"DB_HMI".Bypass_ToolChanger := FALSE;
	"DB_MachineConfig".Bypass_ToolAxis := FALSE;  // Set TRUE if tool axis is not connected
	"DB_MachineConfig".Bypass_MandrelLock := FALSE;  // Set TRUE on variants without MandrelLock cylinder

	// =========================================================================
	// SECTION 10 -- TIMER DEFAULTS
	// â”€â”€â”€â”€â”€â”€â”€â”€â”€â”€â”€â”€â”€â”€â”€â”€â”€â”€â”€â”€â”€â”€â”€â”€â”€â”€â”€â”€â”€â”€â”€â”€â”€â”€â”€â”€â”€â”€â”€â”€â”€â”€â”€â”€â”€â”€â”€â”€â”€â”€â”€â”€â”€â”€â”€â”€â”€â”€â”€â”€â”€â”€â”€â”€â”€â”€â”€â”€â”€â”€â”€â”€â”€
	//  All timer PT values used in the project are set here.
	//  Change a value here to reconfigure every call site at once.
	//  Values revert to these defaults on PLC restart (NON_RETAIN DB).
	// â”€â”€â”€â”€â”€â”€â”€â”€â”€â”€â”€â”€â”€â”€â”€â”€â”€â”€â”€â”€â”€â”€â”€â”€â”€â”€â”€â”€â”€â”€â”€â”€â”€â”€â”€â”€â”€â”€â”€â”€â”€â”€â”€â”€â”€â”€â”€â”€â”€â”€â”€â”€â”€â”€â”€â”€â”€â”€â”€â”€â”€â”€â”€â”€â”€â”€â”€â”€â”€â”€â”€â”€â”€
	//  Cylinder stroke wait times:
	//    Set each slightly above the measured full-stroke time.
	//    No sensor feedback on these â€” machine waits the full duration every cycle.
	// â”€â”€â”€â”€â”€â”€â”€â”€â”€â”€â”€â”€â”€â”€â”€â”€â”€â”€â”€â”€â”€â”€â”€â”€â”€â”€â”€â”€â”€â”€â”€â”€â”€â”€â”€â”€â”€â”€â”€â”€â”€â”€â”€â”€â”€â”€â”€â”€â”€â”€â”€â”€â”€â”€â”€â”€â”€â”€â”€â”€â”€â”€â”€â”€â”€â”€â”€â”€â”€â”€â”€â”€â”€
	//  Process timeouts:
	//    These trigger errors when exceeded; they are safety nets, not normal waits.
	//    Set well above the expected operation time but short enough to catch faults promptly.
	// =========================================================================
	// Cylinder stroke waits
	"DB_MachineConfig".CylMandrelLock_ClampTime := T#0.5S;
	"DB_MachineConfig".CylSheetHolder_RetractTime := T#0.5S;
	"DB_MachineConfig".CylToolHeadLock_PreDelay := T#0.5S;
	"DB_MachineConfig".CylToolHeadLock_RetractTime := T#2S;
	// Process timeouts
	"DB_MachineConfig".Timeout_DriveReady := T#3S;
	"DB_MachineConfig".Timeout_Homing := T#120S;
	"DB_MachineConfig".Timeout_Motion := T#300S;
	"DB_MachineConfig".Timeout_SpindleAtSpeed := T#10S;
	"DB_MachineConfig".Timeout_SpindleStop := T#15S;
	"DB_MachineConfig".Timeout_ToolChange := T#30S;
	"DB_MachineConfig".Timeout_EStopDiscrep := T#500MS;


END_FUNCTION

DATA_BLOCK "TO_AxisSpindle"
{InstructionName := 'TO_PositioningAxis';
 LibVersion := '8.0';
 S7_Optimized_Access := 'TRUE' }
AUTHOR : SIMATIC
FAMILY : BasicMC
NAME : TO_PosAx
VERSION : 8.0
NON_RETAIN
TO_PositioningAxis

BEGIN
   Header.VersionMaj := 8;
   Header.VersionMin := 0;
   Actor.InverseDirection := FALSE;
   Actor.DirectionMode := 1;
   Actor.Interface.EnableDriveOutput.RID := 16#0200_0001;
   Actor.Interface.EnableDriveOutput.AREA := 16#83;
   Actor.Interface.EnableDriveOutput.OFFSET := 10;
   Actor.Interface.PTO := 16#88E1_010C;
   Actor.DriveParameter.PulsesPerDriveRevolution := 500;
   Units.LengthUnit := -1;
   Mechanics.LeadScrew := 1.0;
   DynamicLimits.MaxVelocity := 25000.0;
   DynamicLimits.MinVelocity := 16.66667;
   DynamicDefaults.Acceleration := 24983.33;
   DynamicDefaults.Deceleration := 24983.33;
   DynamicDefaults.EmergencyDeceleration := 12491.67;
   PositionLimits_SW.Active := FALSE;
   PositionLimits_SW.MinPosition := -200.0;
   PositionLimits_SW.MaxPosition := 700.0;
   PositionLimits_HW.Active := FALSE;
   Homing.AutoReversal := FALSE;
   Homing.ApproachDirection := FALSE;
   Homing.ApproachVelocity := 20.0;
   Homing.ReferencingVelocity := 10.0;

END_DATA_BLOCK

DATA_BLOCK "TO_AxisZ"
{InstructionName := 'TO_PositioningAxis';
 LibVersion := '8.0';
 S7_Optimized_Access := 'TRUE' }
AUTHOR : SIMATIC
FAMILY : BasicMC
NAME : TO_PosAx
VERSION : 8.0
NON_RETAIN
TO_PositioningAxis

BEGIN
   Header.VersionMaj := 8;
   Header.VersionMin := 0;
   Actor.InverseDirection := FALSE;
   Actor.Interface.PTO := 16#88E1_010A;
   Actor.DriveParameter.PulsesPerDriveRevolution := 2048;
   Sensor[1].ActiveHoming.DigitalInputAddress.RID := 16#0200_0001;
   Sensor[1].ActiveHoming.DigitalInputAddress.AREA := 16#81;
   Sensor[1].ActiveHoming.DigitalInputAddress.OFFSET := 1;
   Sensor[1].ActiveHoming.HomePositionOffset := 10.0;
   Mechanics.LeadScrew := 1.0;
   DynamicLimits.MaxVelocity := 40.0;
   DynamicLimits.MinVelocity := 0.001;
   DynamicDefaults.Acceleration := 153.8423;
   DynamicDefaults.Deceleration := 184.6107;
   DynamicDefaults.EmergencyDeceleration := 3999.9;
   DynamicDefaults.Jerk := 512.8076;
   PositionLimits_SW.Active := FALSE;
   PositionLimits_SW.MinPosition := -100.0;
   PositionLimits_SW.MaxPosition := 500.0;
   PositionLimits_HW.Active := TRUE;
   PositionLimits_HW.MinSwitchAddress.RID := 16#0200_0001;
   PositionLimits_HW.MinSwitchAddress.AREA := 16#81;
   PositionLimits_HW.MinSwitchAddress.OFFSET := 7;
   PositionLimits_HW.MaxSwitchAddress.RID := 16#0200_0001;
   PositionLimits_HW.MaxSwitchAddress.AREA := 16#81;
   PositionLimits_HW.MaxSwitchAddress.OFFSET := 8;
   Homing.AutoReversal := TRUE;
   Homing.ApproachDirection := FALSE;
   Homing.ApproachVelocity := 30.0;
   Homing.ReferencingVelocity := 10.0;

END_DATA_BLOCK

FUNCTION "FC_ToolAngleCalc" : Void
{ S7_Optimized_Access := 'TRUE' }
VERSION : 0.1
// -----------------------------------------------------------------------------
// FC_ToolAngleCalc -- Automatically calculates tool slot angles based on slot count
//
// When DB_ToolConfig.AutoCalcAngles = TRUE, evenly-spaced angles are calculated
// each scan according to ToolCount:
//   1 slot: [0Â°]
//   2 slot: [0Â°, 180Â°]
//   3 slot: [0Â°, 120Â°, 240Â°]
//   4 slot: [0Â°, 90Â°,  180Â°, 270Â°]
//   General: stepDeg = 360 / ToolCount
//
// When AutoCalcAngles = FALSE, no calculation is performed and Tool1..4_Position
// can be entered manually from the HMI Tool page.
//
// HMI Tool page mapping:
//   DB_MachineConfig.ToolCount        â†’ slot count (1-4, writable)
//   DB_ToolConfig.ToolCode_List[1..4] â†’ slot code (writable, e.g. T101)
//   DB_ToolConfig.Tool1..4_Position   â†’ slot angle (writable when AutoCalcAngles=FALSE)
//   DB_ToolConfig.ToolStepAngle_Calc  â†’ calculated step angle (read-only info)
//   DB_ToolConfig.AutoCalcAngles      â†’ calculation mode (writable)
// -----------------------------------------------------------------------------
   VAR_TEMP
      tc : Int;
      stepDeg : Real;
   END_VAR


BEGIN

	IF NOT "DB_ToolConfig".AutoCalcAngles THEN
	    RETURN;   // Manual mode: do not touch angles
	END_IF;

	// Clamp slot count to 1-4
	#tc := LIMIT(MN := 1, IN := "DB_MachineConfig".ToolCount, MX := 4);
	"DB_MachineConfig".ToolCount := #tc;   // write back clamped value

	// Step angle: 0 for 1 slot (no rotation), equal division for 2+
	IF #tc = 1 THEN
	    #stepDeg := 0.0;
	ELSE
	    #stepDeg := 360.0 / INT_TO_REAL(#tc);
	END_IF;
	"DB_ToolConfig".ToolStepAngle_Calc := #stepDeg;   // for HMI info display

	// Populate slot positions (unused slots remain at 0)
	"DB_ToolConfig".Tool1_Position := 0.0;
	"DB_ToolConfig".Tool2_Position := SEL(G := #tc >= 2, IN0 := 0.0, IN1 := #stepDeg);
	"DB_ToolConfig".Tool3_Position := SEL(G := #tc >= 3, IN0 := 0.0, IN1 := #stepDeg * 2.0);
	"DB_ToolConfig".Tool4_Position := SEL(G := #tc >= 4, IN0 := 0.0, IN1 := #stepDeg * 3.0);

END_FUNCTION

FUNCTION_BLOCK "FB_CylinderControl"
{ S7_Optimized_Access := 'TRUE' }
VERSION : 3.0
// =============================================================================
// FB_CylinderControl -- Pneumatic cylinder control (supports 5/2 and 5/3)
// =============================================================================
//
// â”€â”€â”€ QUICK SETUP â”€â”€â”€â”€â”€â”€â”€â”€â”€â”€â”€â”€â”€â”€â”€â”€â”€â”€â”€â”€â”€â”€â”€â”€â”€â”€â”€â”€â”€â”€â”€â”€â”€â”€â”€â”€â”€â”€â”€â”€â”€â”€â”€â”€â”€â”€â”€â”€â”€â”€â”€â”€â”€â”€â”€â”€â”€â”€â”€â”€â”€
//
//  1) Define physical I/O tags in TIA Portal:
//       "In_Cyl1_AtSetpoint"  Bool  DI   â†’ Mid/target point magnetic switch
//       "In_Cyl1_AtRetract"   Bool  DI   â†’ Retract end magnetic switch (skip if none)
//       "Output_Cyl1_SolA"    Bool  DO   â†’ Solenoid A (extend coil)
//       "Output_Cyl1_SolB"    Bool  DO   â†’ Solenoid B (retract coil, for 5/3)
//
//  2) Call in OB1 in this order (order matters -- sensors must run before cylinder FB):
//       "DB_Sen_Cyl1_Setpt"(RawInput := "In_Cyl1_AtSetpoint");
//       "DB_Sen_Cyl1_Ret"(RawInput   := "In_Cyl1_AtRetract");   // optional
//       "DB_Cylinder1"(
//           SafetyOK       := "Safety_Estop" OR "DB_HMI".Bypass_EStop,
//           Sen_AtSetpoint := "DB_Sen_Cyl1_Setpt".State,
//           Sen_AtRetract  := "DB_Sen_Cyl1_Ret".State
//       );
//       "Output_Cyl1_SolA" := "DB_Cylinder1".Sol_A;
//       "Output_Cyl1_SolB" := "DB_Cylinder1".Sol_B;
//
//  3) Connect DB_Cylinder1 tags in HMI (see table below)
//
//  4) Set DB_Cylinder1.ValveType correctly:
//       2 = 5/3 blocked center  (default, required for ruler mode)
//       1 = 5/2 spring return   (single solenoid, intermediate hold not reliable)
//
// â”€â”€â”€ HMI SCREEN CONNECTIONS â”€â”€â”€â”€â”€â”€â”€â”€â”€â”€â”€â”€â”€â”€â”€â”€â”€â”€â”€â”€â”€â”€â”€â”€â”€â”€â”€â”€â”€â”€â”€â”€â”€â”€â”€â”€â”€â”€â”€â”€â”€â”€â”€â”€â”€â”€â”€â”€â”€â”€
//
//  Writable (HMI â†’ PLC):
//    DB_Cylinder1.Cmd_Extend      Bool   Extend button
//    DB_Cylinder1.Cmd_ExtendFull  Bool   Full extend button -- bypass sensors/ruler; release = stop (pulse use)
//    DB_Cylinder1.Cmd_Retract     Bool   Retract button
//    DB_Cylinder1.Cmd_RetractFull Bool   Full retract button -- bypass sensors/ruler; release = stop (pulse use)
//    DB_Cylinder1.Timeout_Extend  Time   Extend timeout (Modes 0/1/3, default T#5S)
//    DB_Cylinder1.Timeout_Retract Time   Retract timeout (Modes 0/1, default T#5S)
//    DB_Cylinder1.TargetPos       Real   Mode 3: ruler stop position (mm) -- set from HMI or recipe
//    DB_Cylinder1.ValveType       Byte   Valve type (set during commissioning)
//
//  Read-only (PLC â†’ HMI):
//    DB_Cylinder1.State           Int    State code (see STATE CODES)
//    DB_Cylinder1.StateText       String State text
//    DB_Cylinder1.AtSetpoint      Bool   Lamp: locked at setpoint (Modes 0/1)
//    DB_Cylinder1.AtRetract       Bool   Lamp: at retract end (Modes 0/1)
//    DB_Cylinder1.AtTarget        Bool   Lamp: within Tolerance of TargetPos (Mode 2)
//    DB_Cylinder1.PosError        Real   Position error mm (Mode 2)
//    DB_Cylinder1.Error           Bool   Lamp: error present
//    DB_Cylinder1.ErrorID         Word   Error code (display in hex)
//    DB_Cylinder1.Sol_A           Bool   Lamp: SolA energized (for debug)
//    DB_Cylinder1.Sol_B           Bool   Lamp: SolB energized (for debug)
//
//  Sensor status (read-only, for debug screen):
//    DB_Sen_Cyl1_Setpt.State      Bool   Setpoint sensor active?
//    DB_Sen_Cyl1_Ret.State        Bool   Retract end sensor active?
//
// â”€â”€â”€ MANUAL TEST USAGE â”€â”€â”€â”€â”€â”€â”€â”€â”€â”€â”€â”€â”€â”€â”€â”€â”€â”€â”€â”€â”€â”€â”€â”€â”€â”€â”€â”€â”€â”€â”€â”€â”€â”€â”€â”€â”€â”€â”€â”€â”€â”€â”€â”€â”€â”€â”€â”€â”€â”€â”€â”€â”€â”€â”€
//
//  Cylinder FB is called every scan from OB1 -- independent of the state machine.
//  While SafetyOK=TRUE (E-Stop OK or bypass), HMI commands work regardless of
//  whether the machine is in MANUAL, AUTO, or STOPPED mode.
//
//  Test scenarios:
//
//  [A] Full extend (Modes 0/1):
//        Cmd_ExtendFull = TRUE (maintained button)
//        Cylinder extends until Timeout_Extend expires.
//        Returns to Idle when button is released.
//
//  [B] Move to setpoint and hold (5/3 valve, Mode 1):
//        Give Cmd_Extend = TRUE once (momentary sufficient)
//        When Sen_AtSetpoint=TRUE, FB stops and locks. State=3.
//        To retract: Cmd_Retract = TRUE.
//
//  [C] Move to setpoint and hold (5/2 valve, Mode 1):
//        Cmd_Extend = TRUE MUST BE HELD.
//        When Sen_AtSetpoint=TRUE, Sol_A=TRUE is maintained (pressure hold).
//        If button released, spring retracts.
//
//  [D] Retract without sensor (Mode 0):
//        Cmd_Retract = TRUE
//        Transitions to Idle after Timeout_Retract -- no error.
//
//  [E] Ruler zone-pulse positioning (Mode 2, ValveType=2):
//        Set TargetPos (mm). Give Cmd_GotoPos rising edge (or Cmd_Extend/Cmd_Retract).
//        FB fires zone-calculated pulses. Direction auto-selected from PosError sign.
//        After each pulse: solenoid off (mechanical lock) â†’ wait SettleTime â†’ evaluate.
//        Repeats until within Tolerance or MaxCorrections reached (error 16#0505).
//        Each pulse lets the piston travel, then holds; position approaches target step by step.
//
//  [F] Clear error:
//        State=10 (ERROR) â†’ give any command â†’ State=0 (Idle).
//
// â”€â”€â”€ VALVE TYPE SELECTION â”€â”€â”€â”€â”€â”€â”€â”€â”€â”€â”€â”€â”€â”€â”€â”€â”€â”€â”€â”€â”€â”€â”€â”€â”€â”€â”€â”€â”€â”€â”€â”€â”€â”€â”€â”€â”€â”€â”€â”€â”€â”€â”€â”€â”€â”€â”€â”€â”€â”€â”€â”€â”€
//
//  ValveType=1 (5/2 Spring Return):
//    Sol_A=TRUE  â†’ piston extends.  Sol_A=FALSE â†’ piston retracts (spring).
//    Sol_B is never used.
//    âš  On power loss, piston returns to spring position (retracted).
//
//  ValveType=2 (5/3 Blocked Center) -- recommended, required for Mode 2:
//    Sol_A=TRUE, Sol_B=FALSE â†’ extends
//    Sol_A=FALSE, Sol_B=TRUE â†’ retracts
//    Sol_A=FALSE, Sol_B=FALSE â†’ mechanical lock (piston stays in place)
//    âš  On power loss, piston is locked (remains in current position).
//    âš  Purchase BLOCKED CENTER -- do NOT use EXHAUST CENTER (releases on power loss).
//
//  ValveType=3 (5/3 Exhaust Center):
//    Not suitable for holding intermediate positions.
//
// â”€â”€â”€ POSITIONING MODES â”€â”€â”€â”€â”€â”€â”€â”€â”€â”€â”€â”€â”€â”€â”€â”€â”€â”€â”€â”€â”€â”€â”€â”€â”€â”€â”€â”€â”€â”€â”€â”€â”€â”€â”€â”€â”€â”€â”€â”€â”€â”€â”€â”€â”€â”€â”€â”€â”€â”€â”€â”€â”€â”€â”€
//
//  Mode 0 (No sensor):      Cmd_Extend = full stroke; timeout = done, no error.
//  Mode 1 (Magn. switch):   Cmd_Extend waits for Sen_AtSetpoint; timeout = error 16#0501.
//  Mode 2 (Linear ruler):   Zone-pulse positioning. ValveType must be 2.
//                           No digital end sensors used in this mode.
//  Mode 3 (Ruler setpoint): Cmd_Extend/Cmd_GotoPos extends until RulerValue >= TargetPos; solenoid cuts immediately.
//                           TargetPos (mm) is set from HMI (Cyl_TargetPos) or recipe CMD=40 (Param Ã— Cmd40_Gain).
//                           Sol_A held on during extend; solenoid cuts when position reached.
//                           5/3 blocked-center valve recommended (mechanical lock holds position).
//                           RulerValid=FALSE â†’ error 16#0504. Timeout â†’ error 16#0506.
//
// â”€â”€â”€ STATE CODES â”€â”€â”€â”€â”€â”€â”€â”€â”€â”€â”€â”€â”€â”€â”€â”€â”€â”€â”€â”€â”€â”€â”€â”€â”€â”€â”€â”€â”€â”€â”€â”€â”€â”€â”€â”€â”€â”€â”€â”€â”€â”€â”€â”€â”€â”€â”€â”€â”€â”€â”€â”€â”€â”€â”€â”€â”€â”€â”€â”€â”€
//   -1 = E-Stop        SafetyOK=FALSE, all outputs off
//    0 = Idle           No command / waiting
//    1 = Extending      Sol_A=TRUE, waiting for setpoint or timeout (Modes 0/1)
//    2 = Retracting     5/3:Sol_B=TRUE / 5/2:spring (Modes 0/1)
//    3 = At Setpoint    Held at target position, locked (Modes 1/3)
//    4 = At Retract     Retract end sensor triggered (Mode 1)
//    5 = Ruler Pulse    Solenoid firing for zone-calculated duration (Mode 2)
//    7 = Ruler Hold     Both solenoids off (mechanical lock); settles then evaluates (Mode 2)
//   10 = ERROR          Fault condition -- clears on next command
//
// â”€â”€â”€ ERROR CODES â”€â”€â”€â”€â”€â”€â”€â”€â”€â”€â”€â”€â”€â”€â”€â”€â”€â”€â”€â”€â”€â”€â”€â”€â”€â”€â”€â”€â”€â”€â”€â”€â”€â”€â”€â”€â”€â”€â”€â”€â”€â”€â”€â”€â”€â”€â”€â”€â”€â”€â”€â”€â”€â”€â”€â”€â”€â”€â”€â”€â”€
//   16#0501 = Extend timeout   -- Sen_AtSetpoint not received within Timeout_Extend (Mode 1)
//   16#0502 = Retract timeout  -- reserved
//   16#0503 = Sensor conflict        -- Sen_AtSetpoint AND Sen_AtRetract TRUE simultaneously
//   16#0504 = Ruler invalid          -- RulerValid=FALSE during ruler motion (Mode 2)
//   16#0505 = Max corrections        -- MaxCorrections pulses fired without reaching Tolerance (Mode 2)
//   16#0506 = Ruler setpoint timeout -- RulerValue did not reach TargetPos within Timeout_Extend (Mode 3)
//
// â”€â”€â”€ RULER MODE ZONE-PULSE PARAMETERS (Mode 2) â”€â”€â”€â”€â”€â”€â”€â”€â”€â”€â”€â”€â”€â”€â”€â”€â”€â”€â”€â”€â”€â”€â”€â”€â”€â”€â”€â”€â”€â”€â”€
//
//   Zone boundaries are distances from target (mm), all HMI-configurable.
//   The FB selects the pulse duration based on ABS(PosError):
//
//     ABS(PosError) <= Zone1_Limit              â†’ Pulse_Short
//     Zone1_Limit  < ABS(PosError) <= Zone2_Limit â†’ Pulse_Medium
//     Zone2_Limit  < ABS(PosError) <= Zone3_Limit â†’ Pulse_Long
//                    ABS(PosError)  > Zone3_Limit â†’ Pulse_Max
//
//   After each pulse: solenoid off â†’ wait SettleTime â†’ evaluate position â†’ repeat or done.
//   Direction (extend/retract) is auto-selected each pulse from PosError sign.
//   The solenoid is never on longer than the selected pulse duration.
//
// â”€â”€â”€ ADDING A NEW CYLINDER â”€â”€â”€â”€â”€â”€â”€â”€â”€â”€â”€â”€â”€â”€â”€â”€â”€â”€â”€â”€â”€â”€â”€â”€â”€â”€â”€â”€â”€â”€â”€â”€â”€â”€â”€â”€â”€â”€â”€â”€â”€â”€â”€â”€â”€â”€â”€â”€â”€â”€â”€
//   1) Add new instance DBs to 02_DataBlocks.scl:
//        DATA_BLOCK "DB_Cylinder2" ... "FB_CylinderControl"
//        DATA_BLOCK "DB_Sen_Cyl2_Setpt" ... "FB_DigitalSensor"
//   2) Define physical tags in TIA Portal
//   3) Add calls to 08_Main_OB1.scl (sensors before cylinder FB)
//   4) Connect physical outputs: Output_Cyl2_SolA/B := DB_Cylinder2.Sol_A/B
// -----------------------------------------------------------------------------
   VAR_INPUT
      ValveType : Byte := 2;   // 1=5/2_spring  2=5/3_blocked  3=5/3_exhaust Safety -- connected in OB1
      SafetyOK : Bool := FALSE;   // E-Stop OK â†’ output permission Commands -- HMI writes to instance DB, not connected in OB1
      Cmd_Extend : Bool := FALSE;   // Extend: move to setpoint (Mode 1) or TargetPos (Mode 2)
      Cmd_ExtendFull : Bool := FALSE;   // Full extend: bypass sensors/ruler, timeout = done; release = stop (pulse use)
      Cmd_Retract : Bool := FALSE;   // Retract
      Cmd_RetractFull : Bool := FALSE;   // Full retract: bypass sensors/ruler, timeout = done; release = stop (pulse use) Sensor inputs -- connected from FB_DigitalSensor.State in OB1 (Modes 0/1)
      Sen_AtSetpoint : Bool := FALSE;   // Mid/target point magnetic switch (Mode 1)
      Sen_AtRetract : Bool := FALSE;   // Retract end magnetic switch (optional) Timeout -- Modes 0, 1, and 3
      Timeout_Extend : Time := T#5S;
      Timeout_Retract : Time := T#5S;   // Positioning mode -- set from HMI during commissioning 0 = No sensor:     Cmd_Extend acts as full stroke; timeout = done, no error 1 = Magn. switch:  Cmd_Extend waits for Sen_AtSetpoint; timeout = error 16#0501 2 = Linear ruler:  Zone-pulse positioning toward TargetPos; ValveType must be 2 3 = Ruler setpoint: Extend until RulerValue >= TargetPos; solenoid cuts immediately; timeout = error 16#0506
      PositioningMode : Byte := 0;   // Ruler inputs (Modes 2 and 3) -- connect in OB1
      Cmd_GotoPos : Bool := FALSE;   // Rising edge: go to TargetPos (Mode 2 = zone-pulse, Mode 3 = extend until reached)
      RulerValue : Real := 0.0;   // [Modes 2+3] Current position (mm) -- connect to DB_LinearRuler.Value
      RulerValid : Bool := FALSE;   // [Modes 2+3] Measurement valid -- connect to DB_LinearRuler.Valid
      TargetPos : Real := 0.0;   // [Modes 2+3] Target position (mm); clamped by MinPos/MaxPos Ruler position clamp (Modes 2 and 3, 0 = disabled)
      MaxPos : Real := 0.0;   // Max allowed position (mm); clamps TargetPos
      MinPos : Real := 0.0;   // Min allowed position (mm); clamps TargetPos [Mode 2 - Zone-pulse] Accuracy
      Tolerance : Real := 20.0;   // Acceptable position error (mm)
      MaxCorrections : Int := 10;   // Max total pulses before error 16#0505 [Mode 2 - Zone-pulse] Timing
      SettleTime : Time := T#300MS;   // Wait after each pulse before evaluating position [Mode 2 - Zone-pulse] Zone thresholds and pulse durations -- all HMI-configurable Pulse duration is selected by ABS(PosError):   ABS(error) <= Zone1_Limit              â†’ Pulse_Short   (fine correction, near target)   Zone1_Limit < ABS(error) <= Zone2_Limit â†’ Pulse_Medium   Zone2_Limit < ABS(error) <= Zone3_Limit â†’ Pulse_Long                ABS(error)  > Zone3_Limit  â†’ Pulse_Max    (large initial move)
      Zone1_Limit : Real := 10.0;   // [Mode 2 - Zone-pulse] Fine zone boundary (mm)
      Zone2_Limit : Real := 50.0;   // [Mode 2 - Zone-pulse] Medium zone boundary (mm)
      Zone3_Limit : Real := 100.0;   // [Mode 2 - Zone-pulse] Coarse zone boundary (mm)
      Pulse_Short : Time := T#50MS;   // [Mode 2 - Zone-pulse] Finest correction pulse
      Pulse_Medium : Time := T#100MS;   // [Mode 2 - Zone-pulse]
      Pulse_Long : Time := T#250MS;   // [Mode 2 - Zone-pulse]
      Pulse_Max : Time := T#1S;   // [Mode 2 - Zone-pulse] Large initial move pulse
   END_VAR

   VAR_OUTPUT
      Sol_A : Bool;   // Extend solenoid output
      Sol_B : Bool;   // Retract solenoid output (5/3 only)
      State : Int;   // State code
      StateText : String[14];   // HMI state text
      AtSetpoint : Bool;   // Held at setpoint sensor (Modes 0/1)
      AtRetract : Bool;   // Confirmed at retract end (Modes 0/1)
      AtTarget : Bool;   // Mode 2: within Tolerance of TargetPos
      PosError : Real;   // Mode 2: RulerValue - TargetPos (mm)
      Error : Bool;   // Active error
      ErrorID : Word;   // Error code (16#05xx)
   END_VAR

   VAR
      extendFull : Bool;   // ExtendFull mode active (Modes 0/1)
      retractFull : Bool;   // RetractFull mode active
      gotoTargetLatch : Bool;   // GotoPos latch for Mode 3: keeps extending after button release
      tExtend {InstructionName := 'TON_TIME'; LibVersion := '1.0'} : TON_TIME;   // Extend timeout (Modes 0/1/3)
      tRetract {InstructionName := 'TON_TIME'; LibVersion := '1.0'} : TON_TIME;   // Retract timeout (Modes 0/1) Recipe CMD=40 gain: TargetPos = Param Ã— Cmd40_Gain (mm). Set in FC_LoadConfig; adjustable from HMI at runtime.
      Cmd40_Gain : Real := 1.0;
      prevCmdGotoPos : Bool;   // Previous Cmd_GotoPos value (rising edge detection)
      corrAttempts : Int;   // Total pulses fired this move (reset on new command)
      tPulse {InstructionName := 'TON_TIME'; LibVersion := '1.0'} : TON_TIME;   // Mode 2: pulse duration timer (State 5)
      pulseExtend : Bool;   // Mode 2: TRUE = current pulse is extend direction
      calculatedPulse : Time;   // Mode 2: zone-selected pulse duration
      tSettle {InstructionName := 'TON_TIME'; LibVersion := '1.0'} : TON_TIME;   // Mode 2: post-pulse settle timer (State 7)
      inSettling : Bool;   // Mode 2: TRUE = waiting for piston to stop CMD=41 atmosphere override (BackSupport only; unused/FALSE on all other cylinders) Written by FB_RecipeHandler; consumed as OR override in OB1 output assignment.
      SolB_Cmd41 : Bool := FALSE;   // CMD=41 Param=1: hold Sol_B ON independently of state machine
      SolAtmo_Cmd : Bool := FALSE;   // CMD=41 Param=1: ON / Param=2: OFF
   END_VAR

   VAR_TEMP
      effectiveTarget : Real;   // TargetPos clamped to MinPos/MaxPos
      absError : Real;   // ABS(PosError) used for zone selection
   END_VAR


BEGIN

	// â”€â”€ Safety: SafetyOK=FALSE â†’ all outputs off, state=-1 â”€â”€â”€â”€â”€â”€â”€â”€â”€â”€â”€â”€â”€â”€â”€â”€â”€â”€â”€
	IF NOT #SafetyOK THEN
	    #Sol_A := FALSE;
	    #Sol_B := FALSE;
	    #State := -1;
	    #StateText := 'E-Stop';
	    #AtSetpoint := FALSE;
	    #AtRetract := FALSE;
	    RETURN;
	END_IF;

	// â”€â”€ Sensor conflict check (Modes 0/1) â”€â”€â”€â”€â”€â”€â”€â”€â”€â”€â”€â”€â”€â”€â”€â”€â”€â”€â”€â”€â”€â”€â”€â”€â”€â”€â”€â”€â”€â”€â”€â”€â”€â”€â”€â”€
	IF #Sen_AtSetpoint AND #Sen_AtRetract THEN
	    #Sol_A := FALSE;
	    #Sol_B := FALSE;
	    #State := 10;
	    #Error := TRUE;
	    #ErrorID := 16#0503;
	    #StateText := 'ERROR';
	    RETURN;
	END_IF;

	// â”€â”€ Timeout timers (Modes 0/1 only -- States 1 and 2) â”€â”€â”€â”€â”€â”€â”€â”€â”€â”€â”€â”€â”€â”€â”€â”€â”€â”€â”€â”€
	#tExtend(IN := (#State = 1),
	         PT := #Timeout_Extend);
	#tRetract(IN := (#State = 2),
	          PT := #Timeout_Retract);

	// â”€â”€ Effective target: clamp TargetPos to MinPos/MaxPos â”€â”€â”€â”€â”€â”€â”€â”€â”€â”€â”€â”€â”€â”€â”€â”€â”€â”€â”€
	IF #MaxPos > 0.0 AND #TargetPos > #MaxPos THEN
	    #effectiveTarget := #MaxPos;
	ELSIF #MinPos > 0.0 AND #TargetPos < #MinPos THEN
	    #effectiveTarget := #MinPos;
	ELSE
	    #effectiveTarget := #TargetPos;
	END_IF;

	// â”€â”€ State machine â”€â”€â”€â”€â”€â”€â”€â”€â”€â”€â”€â”€â”€â”€â”€â”€â”€â”€â”€â”€â”€â”€â”€â”€â”€â”€â”€â”€â”€â”€â”€â”€â”€â”€â”€â”€â”€â”€â”€â”€â”€â”€â”€â”€â”€â”€â”€â”€â”€â”€â”€â”€â”€â”€â”€â”€â”€
	CASE #State OF

	    -1: // E-Stop cleared â†’ go to Idle
	        #State := 0;

	    0: // IDLE -- waiting for command
	        #Error := FALSE;
	        #ErrorID := 16#0000;
	        #AtTarget := FALSE;
	        #PosError := 0.0;
	        #corrAttempts := 0;
	        #inSettling := FALSE;
	        #gotoTargetLatch := FALSE;

	        IF #Cmd_ExtendFull THEN
	            // Full stroke: ignores all sensors, timeout = mechanical end = done
	            #extendFull := TRUE;
	            #State := 1;

	        ELSIF #Cmd_Extend THEN
	            CASE #PositioningMode OF
	                0: // No sensor -- full stroke
	                    #extendFull := TRUE;
	                    #State := 1;
	                1: // Magnetic switch
	                    #extendFull := FALSE;
	                    #State := 1;
	                2: // Ruler -- zone-pulse toward TargetPos (direction auto-selected)
	                    IF NOT #RulerValid THEN
	                        #State := 10;
	                        #Error := TRUE;
	                        #ErrorID := 16#0504;
	                    ELSE
	                        #State := 5;
	                    END_IF;
	                3: // Ruler setpoint -- extend until RulerValue >= TargetPos
	                    IF NOT #RulerValid THEN
	                        #State := 10;
	                        #Error := TRUE;
	                        #ErrorID := 16#0504;
	                    ELSIF #effectiveTarget > 0.0 AND #RulerValue >= #effectiveTarget THEN
	                        #State := 3;   // Already at or past target position: lock immediately
	                    ELSE
	                        #extendFull := FALSE;
	                        #State := 1;
	                    END_IF;
	                ELSE:
	                    #extendFull := TRUE;
	                    #State := 1;
	            END_CASE;

	        ELSIF #Cmd_Retract THEN
	            IF #PositioningMode = 2 THEN
	                // Ruler mode: zone-pulse toward TargetPos (direction auto-selected)
	                IF NOT #RulerValid THEN
	                    #State := 10;
	                    #Error := TRUE;
	                    #ErrorID := 16#0504;
	                ELSE
	                    #State := 5;
	                END_IF;
	            ELSE
	                #State := 2;
	            END_IF;

	        ELSIF #Cmd_RetractFull THEN
	            // Full retract: bypass all sensors and ruler, retract while held
	            #retractFull := TRUE;
	            #State := 2;

	        ELSIF #Cmd_GotoPos AND NOT #prevCmdGotoPos AND (#PositioningMode = 2 OR #PositioningMode = 3) THEN
	            // Rising edge: go to configured target (Mode 2 = zone-pulse, Mode 3 = extend to level)
	            IF #PositioningMode = 2 THEN
	                IF NOT #RulerValid THEN
	                    #State := 10;
	                    #Error := TRUE;
	                    #ErrorID := 16#0504;
	                ELSIF ABS(#RulerValue - #effectiveTarget) <= #Tolerance THEN
	                    #State := 7;   // Already within tolerance -- lock immediately
	                ELSE
	                    #State := 5;
	                END_IF;
	            ELSE // Mode 3: latched extend to TargetPos
	                IF NOT #RulerValid THEN
	                    #State := 10;
	                    #Error := TRUE;
	                    #ErrorID := 16#0504;
	                ELSIF #effectiveTarget > 0.0 AND #RulerValue >= #effectiveTarget THEN
	                    #State := 3;   // Already at or past target -- lock immediately
	                ELSE
	                    #gotoTargetLatch := TRUE;
	                    #extendFull := FALSE;
	                    #State := 1;
	                END_IF;
	            END_IF;
	        END_IF;
	        #prevCmdGotoPos := #Cmd_GotoPos;

	    1: // EXTENDING -- Sol_A=TRUE, waiting for setpoint or timeout (Modes 0/1/3)
	        IF #PositioningMode = 3 AND NOT #extendFull THEN
	            // Mode 3: watch ruler every scan; cut solenoid when position reached
	            IF NOT #RulerValid THEN
	                #State := 10;
	                #Error := TRUE;
	                #ErrorID := 16#0504;
	            ELSIF #effectiveTarget > 0.0 AND #RulerValue >= #effectiveTarget THEN
	                #State := 3;                  // Position reached: solenoid cuts next scan
	            ELSIF #tExtend.Q THEN
	                #State := 10;
	                #Error := TRUE;
	                #ErrorID := 16#0506;
	            ELSIF NOT #Cmd_Extend AND NOT #Cmd_ExtendFull AND NOT #gotoTargetLatch THEN
	                #State := 0;
	            END_IF;
	        ELSIF #Sen_AtSetpoint AND NOT #extendFull AND #PositioningMode = 1 THEN
	            #State := 3;
	            #extendFull := FALSE;
	        ELSIF #tExtend.Q THEN
	            IF #extendFull THEN
	                // ExtendFull: timeout = mechanical end = success
	                #extendFull := FALSE;
	                #State := 3;
	            ELSE
	                #State := 10;
	                #Error := TRUE;
	                #ErrorID := 16#0501;
	            END_IF;
	        ELSIF NOT #Cmd_Extend AND NOT #Cmd_ExtendFull THEN
	            #State := 0;
	            #extendFull := FALSE;
	        END_IF;

	    2: // RETRACTING -- 5/3:Sol_B=TRUE / 5/2:spring (Modes 0/1)
	        IF #Sen_AtRetract THEN
	            #retractFull := FALSE;
	            #State := 4;
	        ELSIF #tRetract.Q THEN
	            // Timeout = normal completion (no sensor, or sensor absent)
	            #retractFull := FALSE;
	            IF #PositioningMode = 0 THEN
	                #State := 4;   // Mode 0: hold retract solenoid until extend commanded
	            ELSE
	                #State := 0;
	            END_IF;
	        ELSIF NOT #Cmd_Retract AND NOT #Cmd_RetractFull THEN
	            #retractFull := FALSE;
	            #State := 0;
	        END_IF;

	    3: // AT SETPOINT -- held at sensor (Mode 1/3)
	        #gotoTargetLatch := FALSE;
	        IF #Cmd_Retract OR #Cmd_RetractFull THEN
	            #retractFull := #Cmd_RetractFull;
	            #State := 2;
	        ELSIF #Cmd_ExtendFull THEN
	            // Pulse extend from locked position: bypass ruler/sensor
	            #extendFull := TRUE;
	            #State := 1;
	        ELSIF #ValveType = 1 AND NOT #Cmd_Extend AND NOT #Cmd_ExtendFull AND #PositioningMode <> 0 THEN
	            // 5/2: Cmd_Extend released â†’ spring retracts (Mode 0: hold until retract commanded)
	            #State := 2;
	        END_IF;

	    4: // AT RETRACT -- confirmed by Sen_AtRetract=TRUE (Mode 1)
	        IF #Cmd_ExtendFull THEN
	            #extendFull := TRUE;
	            #State := 1;
	        ELSIF #Cmd_Extend THEN
	            CASE #PositioningMode OF
	                0:
	                    #extendFull := TRUE;
	                    #State := 1;
	                1:
	                    #extendFull := FALSE;
	                    #State := 1;
	                2:
	                    IF NOT #RulerValid THEN
	                        #State := 10;
	                        #Error := TRUE;
	                        #ErrorID := 16#0504;
	                    ELSE
	                        #State := 5;
	                    END_IF;
	                3: // Ruler setpoint -- extend until RulerValue >= TargetPos
	                    IF NOT #RulerValid THEN
	                        #State := 10;
	                        #Error := TRUE;
	                        #ErrorID := 16#0504;
	                    ELSIF #effectiveTarget > 0.0 AND #RulerValue >= #effectiveTarget THEN
	                        #State := 3;   // Already at or past target position
	                    ELSE
	                        #extendFull := FALSE;
	                        #State := 1;
	                    END_IF;
	                ELSE:
	                    #extendFull := TRUE;
	                    #State := 1;
	            END_CASE;
	        ELSIF #Cmd_GotoPos AND NOT #prevCmdGotoPos AND (#PositioningMode = 2 OR #PositioningMode = 3) THEN
	            IF #PositioningMode = 2 THEN
	                IF NOT #RulerValid THEN
	                    #State := 10;
	                    #Error := TRUE;
	                    #ErrorID := 16#0504;
	                ELSIF ABS(#RulerValue - #effectiveTarget) <= #Tolerance THEN
	                    #State := 7;
	                ELSE
	                    #corrAttempts := 0;
	                    #State := 5;
	                END_IF;
	            ELSE // Mode 3: latched extend to TargetPos
	                IF NOT #RulerValid THEN
	                    #State := 10;
	                    #Error := TRUE;
	                    #ErrorID := 16#0504;
	                ELSIF #effectiveTarget > 0.0 AND #RulerValue >= #effectiveTarget THEN
	                    #State := 3;
	                ELSE
	                    #gotoTargetLatch := TRUE;
	                    #extendFull := FALSE;
	                    #State := 1;
	                END_IF;
	            END_IF;
	        END_IF;

	    5: // RULER_PULSE -- fires solenoid for zone-calculated duration (Mode 2)
	        //
	        // On first scan in this state (tPulse not yet running):
	        //   1. Calculate PosError and direction (pulseExtend).
	        //   2. Select pulse duration from zone table.
	        //   3. Start tPulse.
	        // On subsequent scans: hold solenoid on until tPulse.Q.
	        // No operator escape during pulse -- SettleTime is short, wait for State 7.
	        // Only exception: ruler loss â†’ immediate fault.
	        IF NOT #RulerValid THEN
	            // Safety: ruler lost during pulse -- cut solenoid and fault
	            #tPulse(IN := FALSE,
	                    PT := T#0ms);
	            #State := 10;
	            #Error := TRUE;
	            #ErrorID := 16#0504;
	        ELSE
	            // Entry: calculate direction and zone-pulse duration
	            IF #tPulse.ET = T#0ms THEN
	                #PosError := #RulerValue - #effectiveTarget;
	                #pulseExtend := #PosError < 0.0;    // undershoot â†’ extend; overshoot â†’ retract
	                #absError := ABS(#PosError);

	                IF #absError <= #Zone1_Limit THEN
	                    #calculatedPulse := #Pulse_Short;
	                ELSIF #absError <= #Zone2_Limit THEN
	                    #calculatedPulse := #Pulse_Medium;
	                ELSIF #absError <= #Zone3_Limit THEN
	                    #calculatedPulse := #Pulse_Long;
	                ELSE
	                    #calculatedPulse := #Pulse_Max;
	                END_IF;
	            END_IF;

	            // Run pulse timer
	            #tPulse(IN := TRUE,
	                    PT := #calculatedPulse);

	            IF #tPulse.Q THEN
	                // Pulse complete: cut solenoid, go to settle + evaluate
	                #tPulse(IN := FALSE,
	                        PT := #calculatedPulse);
	                #corrAttempts := #corrAttempts + 1;
	                #inSettling := TRUE;
	                #State := 7;
	            END_IF;
	        END_IF;

	    7: // RULER_HOLD -- both solenoids off, 5/3 mechanical lock (Mode 2)
	        //
	        // Phase 1 (inSettling=TRUE): wait SettleTime for piston to stop.
	        // Phase 2 (inSettling=FALSE): evaluate position.
	        //   - Within Tolerance â†’ AtTarget=TRUE, hold here.
	        //   - Not at target, pulses remaining â†’ fire next pulse (State 5).
	        //   - Not at target, pulses exhausted â†’ error 16#0505.
	        // Operator commands always take priority in Phase 2.
	        // During Phase 1: wait it out (SettleTime is short).
	        #tSettle(IN := #inSettling,
	                 PT := #SettleTime);
	        IF #tSettle.Q THEN
	            #inSettling := FALSE;
	            #tSettle(IN := FALSE,
	                     PT := #SettleTime);
	        END_IF;

	        IF NOT #inSettling THEN
	            // Phase 2: evaluate position
	            #PosError := #RulerValue - #effectiveTarget;
	            #AtTarget := ABS(#PosError) <= #Tolerance;

	            // Operator commands take priority
	            IF #Cmd_GotoPos AND NOT #prevCmdGotoPos THEN
	                // Re-issue (e.g. TargetPos changed): restart pulse loop
	                IF #RulerValid AND NOT #AtTarget THEN
	                    #corrAttempts := 0;
	                    #inSettling := TRUE;
	                    #State := 5;
	                END_IF;
	            ELSIF #Cmd_ExtendFull THEN
	                // Full stroke override
	                #AtTarget := FALSE;
	                #PosError := 0.0;
	                #corrAttempts := 0;
	                #extendFull := TRUE;
	                #State := 1;
	            ELSIF #Cmd_Retract OR #Cmd_Extend THEN
	                // Manual command while holding: restart toward TargetPos only if not already there
	                IF NOT #AtTarget THEN
	                    #AtTarget := FALSE;
	                    #PosError := 0.0;
	                    #corrAttempts := 0;
	                    #inSettling := TRUE;
	                    #State := 5;
	                END_IF;
	            ELSIF NOT #AtTarget AND #corrAttempts < #MaxCorrections THEN
	                // Auto: fire next correction pulse
	                #inSettling := TRUE;
	                #State := 5;
	            ELSIF NOT #AtTarget AND #corrAttempts >= #MaxCorrections THEN
	                #State := 10;
	                #Error := TRUE;
	                #ErrorID := 16#0505;
	            END_IF;
	        END_IF;

	    10: // ERROR -- clears on any new command, on GotoPos retry, or auto-clears when
	        // idle (no command held). The idle auto-clear prevents a stale cylinder error
	        // (e.g. from an extend timeout) from blocking the next machine run without
	        // requiring the operator to press E-Stop to cycle SafetyOK.
	        IF #Cmd_Extend OR #Cmd_ExtendFull OR #Cmd_Retract OR #Cmd_RetractFull THEN
	            #Error := FALSE;
	            #ErrorID := 16#0000;
	            #State := 0;
	        ELSIF #Cmd_GotoPos AND NOT #prevCmdGotoPos AND (#PositioningMode = 2 OR #PositioningMode = 3) THEN
	            // GotoPos rising edge clears error and restarts motion
	            #Error := FALSE;
	            #ErrorID := 16#0000;
	            #corrAttempts := 0;
	            IF #PositioningMode = 2 THEN
	                IF NOT #RulerValid THEN
	                    #State := 10;
	                    #Error := TRUE;
	                    #ErrorID := 16#0504;
	                ELSIF ABS(#RulerValue - #effectiveTarget) <= #Tolerance THEN
	                    #State := 7;
	                ELSE
	                    #State := 5;
	                END_IF;
	            ELSE // Mode 3
	                IF NOT #RulerValid THEN
	                    #State := 10;
	                    #Error := TRUE;
	                    #ErrorID := 16#0504;
	                ELSIF #effectiveTarget > 0.0 AND #RulerValue >= #effectiveTarget THEN
	                    #State := 3;
	                ELSE
	                    #gotoTargetLatch := TRUE;
	                    #extendFull := FALSE;
	                    #State := 1;
	                END_IF;
	            END_IF;
	        ELSE
	            // No command held and no GotoPos request: auto-clear to IDLE.
	            // The cylinder will retry normally on the next Cmd_Extend.
	            #Error := FALSE;
	            #ErrorID := 16#0000;
	            #State := 0;
	        END_IF;

	    ELSE
	        #State := 0;

	END_CASE;

	// â”€â”€ Solenoid outputs â”€â”€â”€â”€â”€â”€â”€â”€â”€â”€â”€â”€â”€â”€â”€â”€â”€â”€â”€â”€â”€â”€â”€â”€â”€â”€â”€â”€â”€â”€â”€â”€â”€â”€â”€â”€â”€â”€â”€â”€â”€â”€â”€â”€â”€â”€â”€â”€â”€â”€â”€â”€â”€â”€
	CASE #State OF
	    1: // EXTENDING (Modes 0/1)
	        #Sol_A := TRUE;
	        #Sol_B := FALSE;
	    2: // RETRACTING (Modes 0/1)
	        IF #ValveType = 1 THEN
	            #Sol_A := FALSE;
	            #Sol_B := FALSE;
	        ELSE
	            #Sol_A := FALSE;
	            #Sol_B := TRUE;
	        END_IF;
	    3: // AT SETPOINT (Mode 0/1/3)
	        IF #PositioningMode = 0 THEN
	            #Sol_A := TRUE;                              // Mode 0: hold until retract commanded
	            #Sol_B := FALSE;
	        ELSIF #ValveType = 1 THEN
	            #Sol_A := #Cmd_Extend OR #Cmd_ExtendFull;   // pressure hold
	            #Sol_B := FALSE;
	        ELSE
	            #Sol_A := FALSE;                             // 5/3 blocked: mechanical lock
	            #Sol_B := FALSE;
	        END_IF;
	    5: // RULER_PULSE: fire in zone-calculated direction (Mode 2)
	        IF #pulseExtend THEN
	            #Sol_A := TRUE;
	            #Sol_B := FALSE;
	        ELSE
	            #Sol_A := FALSE;
	            #Sol_B := TRUE;     // 5/3 blocked: active retract
	        END_IF;
	    4: // AT RETRACT (Mode 0/1)
	        IF #PositioningMode = 0 AND #ValveType <> 1 THEN
	            #Sol_A := FALSE;
	            #Sol_B := TRUE;                              // Mode 0 + 5/3: hold retract solenoid
	        ELSE
	            #Sol_A := FALSE;                             // Mode 1 or 5/2: both off
	            #Sol_B := FALSE;
	        END_IF;
	    7: // RULER_HOLD: mechanical lock (Mode 2)
	        #Sol_A := FALSE;
	        #Sol_B := FALSE;
	    ELSE
	        // IDLE, E-STOP, ERROR: both off
	        #Sol_A := FALSE;
	        #Sol_B := FALSE;
	END_CASE;

	// â”€â”€ Edge latch for Cmd_GotoPos -- updated every scan after state machine â”€â”€
	#prevCmdGotoPos := #Cmd_GotoPos;

	// â”€â”€ State text â”€â”€â”€â”€â”€â”€â”€â”€â”€â”€â”€â”€â”€â”€â”€â”€â”€â”€â”€â”€â”€â”€â”€â”€â”€â”€â”€â”€â”€â”€â”€â”€â”€â”€â”€â”€â”€â”€â”€â”€â”€â”€â”€â”€â”€â”€â”€â”€â”€â”€â”€â”€â”€â”€â”€â”€â”€â”€â”€â”€
	CASE #State OF
	    -1:
	        #StateText := 'E-Stop';
	    0:
	        #StateText := 'Idle';
	    1:
	        IF #extendFull THEN
	            #StateText := 'Extend Full';
	        ELSE
	            #StateText := 'Extending';
	        END_IF;
	    2:
	        IF #retractFull THEN
	            #StateText := 'Retract Full';
	        ELSE
	            #StateText := 'Retracting';
	        END_IF;
	    3:
	        #StateText := 'At Setpoint';
	    4:
	        #StateText := 'At Retract';
	    5:
	        IF #pulseExtend THEN
	            #StateText := 'Pulse Extend';
	        ELSE
	            #StateText := 'Pulse Retract';
	        END_IF;
	    7:
	        #StateText := 'Ruler Hold';
	    10:
	        #StateText := 'ERROR';
	    ELSE:
	        #StateText := '?';
	END_CASE;

	// â”€â”€ Position confirmation outputs â”€â”€â”€â”€â”€â”€â”€â”€â”€â”€â”€â”€â”€â”€â”€â”€â”€â”€â”€â”€â”€â”€â”€â”€â”€â”€â”€â”€â”€â”€â”€â”€â”€â”€â”€â”€â”€â”€â”€â”€â”€
	#AtSetpoint := (#State = 3);
	#AtRetract := (#State = 4);
	// AtTarget and PosError are updated continuously in State 7 (RULER_HOLD)

END_FUNCTION_BLOCK

FUNCTION_BLOCK "FB_Process"
{ S7_Optimized_Access := 'TRUE' }
VERSION : 4.0
// -----------------------------------------------------------------------------
// FB_Process - Main supervisory state machine with PRE-SCAN
// -----------------------------------------------------------------------------
   VAR_INPUT
      Panel_Start : Bool;
      Panel_Stop : Bool;
      Panel_Pause : Bool;
      Panel_Reset : Bool;
      Rem_Start : Bool;
      Rem_Stop : Bool;
      EStop_OK : Bool := TRUE;   // NC limit switches (FALSE = limit hit, fail-safe)
      Door_Closed : Bool := TRUE;
      AirPressure_OK : Bool := TRUE;
      HW_NC_X_Min : Bool;   // PNP NO proximity sensors (TRUE = limit zone, pre-warning before NC)
      HW_NC_X_Max : Bool;
      HW_NC_Z_Min : Bool;
      HW_NC_Z_Max : Bool;
      HW_PNP_X_Min : Bool;
      HW_PNP_X_Max : Bool;
      HW_PNP_Z_Min : Bool;
      HW_PNP_Z_Max : Bool;
   END_VAR

   VAR_OUTPUT
      Running : Bool;
      IsPaused : Bool;
      Error : Bool;
      StatusID : Int;
      CurrentTool : Int;
      SafeToRun : Bool;
   END_VAR

   VAR_IN_OUT
      Axis_X {InstructionName := 'TO_PositioningAxis'; LibVersion := '8.0'} : TO_PositioningAxis;
      Axis_Z {InstructionName := 'TO_PositioningAxis'; LibVersion := '8.0'} : TO_PositioningAxis;
      Axis_Tool {InstructionName := 'TO_PositioningAxis'; LibVersion := '8.0'} : TO_PositioningAxis;
      Axis_Spindle {InstructionName := 'TO_PositioningAxis'; LibVersion := '8.0'} : TO_PositioningAxis;
   END_VAR

   VAR
      State : Int;   // Recipe handlers (one per program for flexibility)
      fbRecipeHandler : "FB_RecipeHandler";
      fbPreScan : "FB_RecipePreScan";   // Support FBs
      fbToolChanger : "FB_ToolChanger";
      fbHomeX : "FB_Axis_Home";
      fbHomeZ : "FB_Axis_Home";
      fbHomeTool : "FB_Axis_Home";
      fbSpindleControl : "FB_SpindleControl";
      fbManualMode : "FB_ManualMode";
      fbPowerX : "FB_Axis_Power";
      fbPowerZ : "FB_Axis_Power";
      fbPowerTool : "FB_Axis_Power";
      fbResetX : "FB_Axis_Reset";
      fbResetZ : "FB_Axis_Reset";
      fbResetTool : "FB_Axis_Reset";
      fbResetSpindle : "FB_Axis_Reset";
      fbInputs : "FB_InputManager";
      fbLimitMonitor : "FB_LimitMonitor";
      fbSafetyMonitor : "FB_SafetyMonitor";
      fbAlarmManager : "FB_AlarmManager";   // Additional motion FBs for moving to position 0 after stop
      fbMoveX_Stop : "FB_Axis_AbsPos";   // Homing clearance moves (pre + post homing)
      fbMoveZ_Stop : "FB_Axis_AbsPos";   // Homing clearance moves (pre + post homing)
      fbMoveX_HomeClr : "FB_Axis_AbsPos";
      fbMoveZ_HomeClr : "FB_Axis_AbsPos";
      bHomeClrX : Bool;   // PNP proximity sensor halt: controlled stop when PNP zone entered in auto mode
      bHomeClrZ : Bool;   // PNP proximity sensor halt: controlled stop when PNP zone entered in auto mode
      fbHaltX_PNP : "FB_Axis_Halt";
      fbHaltZ_PNP : "FB_Axis_Halt";
      bHaltX_PNP : Bool;   // Halt execute flags (cleared when state returns to STOPPED) ITEM-31: reset/startup halt â€” aborts any MC_Home the TO may resume after drive power-cycle or warm restart
      bHaltZ_PNP : Bool;   // Halt execute flags (cleared when state returns to STOPPED) ITEM-31: reset/startup halt â€” aborts any MC_Home the TO may resume after drive power-cycle or warm restart
      fbHaltX_Reset : "FB_Axis_Halt";
      fbHaltZ_Reset : "FB_Axis_Halt";
      fbHaltTool_Reset : "FB_Axis_Halt";
      bHaltAllAxes : Bool;   // Pulse: TRUE for one scan; set by bDoHardReset + first-scan startup; cleared after FB calls Control flags
      bPreScanExec : Bool;
      bResetRecipe : Bool;   // One-shot flag to reset FB_RecipeHandler
      bStartSeq : Bool;
      bToolExecute : Bool;
      bPauseActive : Bool;
      bStopMoveX : Bool;   // Flags for moving to position 0 after stop Sequential homing (startup): home X then Z then Tool in active mode (mode 3)
      bStopMoveZ : Bool;   // Flags for moving to position 0 after stop Sequential homing (startup): home X then Z then Tool in active mode (mode 3)
      bHomeXExec : Bool;
      bHomeZExec : Bool;
      bHomeToolExec : Bool;
      homeSeqState : Int;   // 0=idle, 1=homing X, 2=homing Z, 3=homing Tool
      activeToolReq : Int;
      activeToolDone : Bool;
      newErrorFlag : Bool;
      newErrorCode : Word;
      bSpindleStart : Bool;
      bSpindleStop : Bool;
      bDrivesEnable : Bool;
      prevAckError : Bool;
      prevRestart : Bool;
      prevContinue : Bool;
      ackEdge : Bool;
      restartEdge : Bool;
      continueEdge : Bool;
      prevApplyToolConfig : Bool;   // previous ApplyToolConfig button state
      applyToolEdge : Bool;   // rising edge for apply tool mapping
      prevProdReset : Bool;
      prevLastCycleReset : Bool;
      prodResetEdge : Bool;
      lastCycleResetEdge : Bool;
      prevSafetyError : Bool;
      prevDriveFaultX : Bool;   // Edge detection: X drive power failure
      prevDriveFaultZ : Bool;   // Edge detection: Z drive power failure
      prevDriveFaultTool : Bool;   // ITEM-29: edge detection: tool axis drive power failure
      prevTOFaultX : Bool;   // Edge detection: X axis TO fault (StatusBits.Error poller)
      prevTOFaultZ : Bool;   // Edge detection: Z axis TO fault
      prevTOFaultTool : Bool;   // Edge detection: Tool axis TO fault
      prevTOFaultSpindle : Bool;   // Edge detection: Spindle TO fault
      bJogBlockPlus : Bool;   // Manual soft-limit jog gate: block jog+ (recomputed every scan)
      bJogBlockMinus : Bool;   // Manual soft-limit jog gate: block jog- (recomputed every scan)
      prevManualError : Bool;   // Edge detection: manual mode error
      bInitDone : Bool;   // TRUE after first PLC scan; prevents re-triggering startup reset
      bDoHardReset : Bool;   // Pulse: set TRUE to trigger hard-reset block this scan (startup + Cmd_Reset)
      applyIndex : Int;   // Loop index for tool config apply Active recipe reference
      activeProgram : Int;
      activeLineCount : Int;   // ToolHeadLock timers
      tonLockWait {InstructionName := 'TON_TIME'; LibVersion := '1.0'} : TON_TIME;   // Fallback timeout for states 17 and 29 (T#3S)
      tonLockPreDelay {InstructionName := 'TON_TIME'; LibVersion := '1.0'} : TON_TIME;   // Pre-delay before commanding extend in state 17 (T#1S) TRUE = LOCK_RETRACT_WAIT exits to STATE_STOPPED (axes already at zero from STOPPING) FALSE = exits to STATE_TOOL_CHANGE
      bLockAfterHoming : Bool;   // Sheet wait (STATE_SHEET_WAIT = 14)
      bSheetWaitPhase2 : Bool;   // Phase 2: MandrelLock extending (T#5S)
      bSheetWaitPhase3 : Bool;   // Phase 3: SheetHolder retracting (T#5S)
      tonMandrelWait {InstructionName := 'TON_TIME'; LibVersion := '1.0'} : TON_TIME;   // T#5S open-loop stroke wait for MandrelLock (phase 2)
      tonSheetHolderRetract {InstructionName := 'TON_TIME'; LibVersion := '1.0'} : TON_TIME;   // T#5S open-loop wait for SheetHolder retract (phase 3)
      bMandrelRetractPulse : Bool;   // One-shot: pulse Cmd_Retract for one scan to release MandrelLock FB from State 3
      bMandrelRetractPending : Bool;   // ITEM-32: deferred retract â€” unsafe paths (Reset/Error/Complete) set this; SpindleStopSafeTime timer promotes to pulse
      tonMandrelRetractWait {InstructionName := 'TON_TIME'; LibVersion := '1.0'} : TON_TIME;   // ITEM-32: safety gate timer for deferred retract (PT = DB_MachineConfig.SpindleStopSafeTime)
      bSheetHolderRetractPulse : Bool;   // One-shot: pulse Cmd_Retract for one scan to release SheetHolder FB from State 3
      bWaitingSpindleStop : Bool;   // TRUE while STATE_STOPPING waits for spindle decel before retracting MandrelLock
      tonSpindleStopWait {InstructionName := 'TON_TIME'; LibVersion := '1.0'} : TON_TIME;   // Proportional wait before MandrelLock retract (see SpindleStopSafeTime). Fires immediately if speed was 0.
      capturedSpindleRPM : Real;   // Speed captured when bWaitingSpindleStop is set (ITEM-28)
      spindleStopPT : Time;   // Proportional PT for tonSpindleStopWait (ITEM-28)
      bCycleCountDone : Bool;   // One-shot: prevents multiple CycleCount increments per cycle (ITEM-20) Cycle timer
      tonElapsed {InstructionName := 'TON_TIME'; LibVersion := '1.0'} : TON_TIME;   // Homing timeout: fires if STATE_HOMING sequence takes longer than 120s
      tonHomingTimeout {InstructionName := 'TON_TIME'; LibVersion := '1.0'} : TON_TIME;   // ITEM-30: independent timeout for STATE_STOP_GOHOME (was sharing tonHomingTimeout â€” risky if a normal homing cycle consumed most of the budget, leaving too little time for post-stop homing)
      tonStopHomeTimeout {InstructionName := 'TON_TIME'; LibVersion := '1.0'} : TON_TIME;   // Drive ready timeout: fires if drives do not become ready within 3s of STATE_STARTING
      tonDriveReady {InstructionName := 'TON_TIME'; LibVersion := '1.0'} : TON_TIME;   // Spindle deceleration wait
      tonSpindleDecel {InstructionName := 'TON_TIME'; LibVersion := '1.0'} : TON_TIME;   // Decel wait timer
      bSpindleDecelWait : Bool;   // TRUE while waiting for decel to complete
      bSpindlePendingStart : Bool;   // Deferred start captured during decel wait
      pendingSpindleSpeed : Real;   // Speed to apply when timer expires
      elapsedAccum : Time;   // Accumulated elapsed time
      timerRunning : Bool;   // Timer active flag
      elapsedSeconds : DInt;   // Seconds counter Warm restart
      savedLineIndex : Int := -1;   // Saved line for restart (-1 = none)
      savedProgram : Int := -1;   // Saved program for restart Production logging
      prevState : Int;   // For state edge detection
      prodTimeNow {InstructionName := 'DTL'; LibVersion := '1.0'} : DTL;
      prodTimeStatus : Int;   // Spindle history ring buffer: previous values for change detection A new snapshot is pushed only when one of these changes.
      prevSnap_State : Int;
      prevSnap_PrevStart : Bool;
      prevSnap_ReqStart : Bool;
      prevSnap_StartEdge : Bool;
      prevSnap_MoveVelBusy : Bool;   // MC_MoveVelocity.Busy -- triggers snapshot when TO accepts/drops command
   END_VAR

   VAR CONSTANT
      STATE_STOPPED : Int := 0;
      STATE_MANUAL : Int := 5;
      STATE_STARTING : Int := 10;
      STATE_PRE_SCAN : Int := 12;
      STATE_PRE_HOME_CLR : Int := 13;   // Pre-homing clearance move out of PNP zone
      STATE_SHEET_WAIT : Int := 14;   // Sheet insertion: Ph1=SheetHolder extends+prompt, Ph2=MandrelLock T#5S, Ph3=SheetHolder retract T#5S â†’ LOCK_EXTEND_WAIT
      STATE_HOMING : Int := 15;
      STATE_POST_HOME_CLR : Int := 16;   // Post-homing clearance move away from PNP zone
      STATE_STOPPING : Int := 18;
      STATE_STOP_GOHOME : Int := 19;
      STATE_STOP_GOTOZERO : Int := 21;
      STATE_PNP_HALT : Int := 22;   // PNP limit zone -- halt active, reverse jog allowed
      STATE_RUNNING : Int := 20;
      STATE_PAUSED : Int := 25;
      STATE_TOOL_CHANGE : Int := 30;
      STATE_TOOL_WAIT : Int := 35;
      STATE_LOCK_EXTEND_WAIT : Int := 17;   // ToolHeadLock engaging before RUNNING
      STATE_LOCK_RETRACT_WAIT : Int := 29;   // ToolHeadLock releasing before tool change or homing
      STATE_ERROR : Int := 999;
   END_VAR


BEGIN

	// Update HMI displays
	"DB_HMI".ActualX := #Axis_X.ActualPosition;
	"DB_HMI".ActualZ := #Axis_Z.ActualPosition;
	"DB_HMI".MachineState := #State;

	// =========================================================================
	// FIRST-SCAN STARTUP INIT
	// =========================================================================
	// On the very first PLC scan after power-up or warm restart, trigger a hard
	// reset. This forces a known-clean machine state explicitly rather than
	// relying solely on NON_RETAIN default values. Covers any case where the
	// state machine variable did not reset cleanly (e.g. mid-homing on restart).
	IF NOT #bInitDone THEN
	    #bDoHardReset := TRUE;
	    #bHaltAllAxes := TRUE;   // ITEM-31: abort any MC_Home the TO may auto-resume on power-up
	    #bInitDone := TRUE;
	END_IF;

	// Edge detection for buttons
	#ackEdge := "DB_HMI".Btn_AckError AND NOT #prevAckError;
	#prevAckError := "DB_HMI".Btn_AckError;
	#restartEdge := "DB_HMI".Btn_Restart AND NOT #prevRestart;
	#prevRestart := "DB_HMI".Btn_Restart;
	#continueEdge := "DB_HMI".Btn_Continue AND NOT #prevContinue;
	#prevContinue := "DB_HMI".Btn_Continue;
	// Apply Tool Config edge
	#applyToolEdge := "DB_HMI".Btn_ApplyToolConfig AND NOT #prevApplyToolConfig;
	#prevApplyToolConfig := "DB_HMI".Btn_ApplyToolConfig;
	#prodResetEdge := "DB_HMI".Btn_ProdReset AND NOT #prevProdReset;
	#prevProdReset := "DB_HMI".Btn_ProdReset;
	#lastCycleResetEdge := "DB_HMI".Btn_LastCycleReset AND NOT #prevLastCycleReset;
	#prevLastCycleReset := "DB_HMI".Btn_LastCycleReset;

	// Get active program from HMI (lock during RUNNING to prevent mid-program switch)
	IF #State < #STATE_STARTING OR #State >= #STATE_ERROR THEN
	    #activeProgram := "DB_HMI".ProductSelect;
	    IF #activeProgram < 1 THEN
	        #activeProgram := 1;
	    END_IF;
	    IF #activeProgram > 5 THEN
	        #activeProgram := 5;
	    END_IF;
	END_IF;

	// Apply tool-slot mapping from HMI -> DB_ToolConfig when operator requests it.
	IF #applyToolEdge THEN
	    // Only copy up to 4 slots; respect configured ToolCount
	    FOR #applyIndex := 1 TO 4 DO
	        IF #applyIndex <= "DB_MachineConfig".ToolCount THEN
	            "DB_ToolConfig".ToolCode_List[#applyIndex] := "DB_HMI".ToolSlotCode[#applyIndex];
	        END_IF;
	    END_FOR;
	END_IF;

	// Safety monitor
	#fbSafetyMonitor(EStop_OK := #EStop_OK,
	                 Door_Closed := #Door_Closed,
	                 AirPressure_OK := #AirPressure_OK,
	                 DrivesReady := #fbPowerX.Status AND #fbPowerZ.Status,
	                 Bypass_EStop := "DB_HMI".Bypass_EStop,
	                 Bypass_Door := "DB_HMI".Bypass_Door,
	                 Bypass_AirPressure := "DB_HMI".Bypass_AirPressure,
	                 Bypass_Drives := "DB_HMI".Bypass_Drives);

	// Power control
	#bDrivesEnable := (#EStop_OK OR "DB_HMI".Bypass_EStop) AND (#State <> #STATE_ERROR);
	#fbPowerX(Enable := #bDrivesEnable,
	          Axis := #Axis_X);
	#fbPowerZ(Enable := #bDrivesEnable,
	          Axis := #Axis_Z);
	#fbPowerTool(Enable := #bDrivesEnable AND NOT "DB_MachineConfig".Bypass_ToolAxis,
	             Axis := #Axis_Tool);

	// Drive power failure detection -- capture TO ErrorID and write to diagnostic
	// Checked every scan; alarm is raised only when a new error occurs (rising edge).
	// STATE_PRE_SCAN(12) is treated like STATE_STOPPED(0): contactors are still open during
	// pre-scan (closed only in STATE_STARTING), so a drive fault here is typically a latched
	// fault from a previous run or a transient after TO reset -- not a new startup failure.
	// The drive ready check (tonDriveReady) and MC_Home.Error in STATE_STARTING handle genuine
	// startup faults. Firing STATE_ERROR in PRE_SCAN would abort the recipe validation for no reason.
	IF #fbPowerX.Error THEN
	    "DB_Diagnostic".Power_X_ErrorID := #fbPowerX.ErrorID;
	    "DB_Diagnostic".TO_ErrorText := "FC_TO_ErrorText"(Code := #fbPowerX.ErrorID);
	    IF NOT #prevDriveFaultX THEN
	        #newErrorFlag := TRUE;
	        #newErrorCode := 16#0009;
	        "DB_HMI".ErrorDetail := CONCAT(IN1 := 'TO:', IN2 := "DB_Diagnostic".TO_ErrorText);
	        "DB_HMI".ErrorDetail_ES := CONCAT(IN1 := 'TO:', IN2 := "DB_Diagnostic".TO_ErrorText);
	        IF #State <> #STATE_ERROR AND #State <> 0 AND #State <> #STATE_PRE_SCAN THEN
	            #State := #STATE_ERROR;
	        END_IF;
	    END_IF;
	    #prevDriveFaultX := TRUE;
	ELSE
	    #prevDriveFaultX := FALSE;
	END_IF;

	IF #fbPowerZ.Error THEN
	    "DB_Diagnostic".Power_Z_ErrorID := #fbPowerZ.ErrorID;
	    "DB_Diagnostic".TO_ErrorText := "FC_TO_ErrorText"(Code := #fbPowerZ.ErrorID);
	    IF NOT #prevDriveFaultZ THEN
	        #newErrorFlag := TRUE;
	        #newErrorCode := 16#000A;
	        "DB_HMI".ErrorDetail := CONCAT(IN1 := 'TO:', IN2 := "DB_Diagnostic".TO_ErrorText);
	        "DB_HMI".ErrorDetail_ES := CONCAT(IN1 := 'TO:', IN2 := "DB_Diagnostic".TO_ErrorText);
	        IF #State <> #STATE_ERROR AND #State <> 0 AND #State <> #STATE_PRE_SCAN THEN
	            #State := #STATE_ERROR;
	        END_IF;
	    END_IF;
	    #prevDriveFaultZ := TRUE;
	ELSE
	    #prevDriveFaultZ := FALSE;
	END_IF;

	// ITEM-29: tool axis drive power fault monitoring (mirrors X/Z pattern above)
	IF #fbPowerTool.Error THEN
	    "DB_Diagnostic".TO_ErrorText := "FC_TO_ErrorText"(Code := #fbPowerTool.ErrorID);
	    IF NOT #prevDriveFaultTool THEN
	        #newErrorFlag := TRUE;
	        #newErrorCode := 16#000D;
	        "DB_HMI".ErrorDetail := CONCAT(IN1 := 'TO:', IN2 := "DB_Diagnostic".TO_ErrorText);
	        "DB_HMI".ErrorDetail_ES := CONCAT(IN1 := 'TO:', IN2 := "DB_Diagnostic".TO_ErrorText);
	        IF #State <> #STATE_ERROR AND #State <> 0 AND #State <> #STATE_PRE_SCAN THEN
	            #State := #STATE_ERROR;
	        END_IF;
	    END_IF;
	    #prevDriveFaultTool := TRUE;
	ELSE
	    #prevDriveFaultTool := FALSE;
	END_IF;

	// =========================================================================
	// TO (Technology Object) FAULT POLLER
	// =========================================================================
	// Guarantees axis TO errors ALWAYS reach the HMI. The MC_ wrapper FBs only report
	// an ErrorID while their own command is active; a TO fault outside an active command
	// (following error, TO-internal soft-limit trip, encoder/drive fault at rest) was
	// previously visible only on the TIA Portal TO diagnostics page.
	// Polls <axis>.StatusBits.Error every scan, raises a motion-tier alarm on the rising
	// edge. Skipped while the matching MC_Power FB reports a fault (the drive-power blocks
	// above already raise the more specific 16#0009/16#000A/16#000D) and while E-Stop is
	// active (the safety tier owns that case; power removal marks every axis in error).
	// TO errors are cleared by the MC_Reset calls on AckError/Reset (fbResetX/Z/Tool/Spindle).
	IF #Axis_X.StatusBits.Error AND NOT #fbPowerX.Error AND #EStop_OK THEN
	    IF NOT #prevTOFaultX THEN
	        #newErrorFlag := TRUE;
	        #newErrorCode := 16#0021;
	        "DB_Diagnostic".Error_Text := 'TO fault: X axis (StatusBits.Error) - check TO diagnostics';
	        "DB_HMI".ErrorDetail := 'X axis technology object fault - press Ack/Reset to clear';
	        "DB_HMI".ErrorDetail_ES := 'Fallo de objeto tecnologico eje X - presionar Ack/Reset para borrar';
	        IF #State <> #STATE_ERROR AND #State <> 0 AND #State <> #STATE_PRE_SCAN THEN
	            #State := #STATE_ERROR;
	        END_IF;
	    END_IF;
	    #prevTOFaultX := TRUE;
	ELSE
	    #prevTOFaultX := FALSE;
	END_IF;

	IF #Axis_Z.StatusBits.Error AND NOT #fbPowerZ.Error AND #EStop_OK THEN
	    IF NOT #prevTOFaultZ THEN
	        #newErrorFlag := TRUE;
	        #newErrorCode := 16#0022;
	        "DB_Diagnostic".Error_Text := 'TO fault: Z axis (StatusBits.Error) - check TO diagnostics';
	        "DB_HMI".ErrorDetail := 'Z axis technology object fault - press Ack/Reset to clear';
	        "DB_HMI".ErrorDetail_ES := 'Fallo de objeto tecnologico eje Z - presionar Ack/Reset para borrar';
	        IF #State <> #STATE_ERROR AND #State <> 0 AND #State <> #STATE_PRE_SCAN THEN
	            #State := #STATE_ERROR;
	        END_IF;
	    END_IF;
	    #prevTOFaultZ := TRUE;
	ELSE
	    #prevTOFaultZ := FALSE;
	END_IF;

	IF #Axis_Tool.StatusBits.Error AND NOT #fbPowerTool.Error AND #EStop_OK
	    AND NOT "DB_MachineConfig".Bypass_ToolAxis THEN
	    IF NOT #prevTOFaultTool THEN
	        #newErrorFlag := TRUE;
	        #newErrorCode := 16#0023;
	        "DB_Diagnostic".Error_Text := 'TO fault: Tool axis (StatusBits.Error) - check TO diagnostics';
	        "DB_HMI".ErrorDetail := 'Tool axis technology object fault - press Ack/Reset to clear';
	        "DB_HMI".ErrorDetail_ES := 'Fallo de objeto tecnologico eje herramienta - presionar Ack/Reset para borrar';
	        IF #State <> #STATE_ERROR AND #State <> 0 AND #State <> #STATE_PRE_SCAN THEN
	            #State := #STATE_ERROR;
	        END_IF;
	    END_IF;
	    #prevTOFaultTool := TRUE;
	ELSE
	    #prevTOFaultTool := FALSE;
	END_IF;

	// Spindle: MC_Power lives inside fbSpindleControl (no fbPowerSpindle guard here).
	// A same-scan specific spindle error (16#05xx) from FB_SpindleControl wins the display
	// anyway (same tier, first-in latch); this poller is the safety net for faults at rest.
	IF #Axis_Spindle.StatusBits.Error AND #EStop_OK THEN
	    IF NOT #prevTOFaultSpindle THEN
	        #newErrorFlag := TRUE;
	        #newErrorCode := 16#0024;
	        "DB_Diagnostic".Error_Text := 'TO fault: Spindle (StatusBits.Error) - check TO diagnostics';
	        "DB_HMI".ErrorDetail := 'Spindle technology object fault - press Ack/Reset to clear';
	        "DB_HMI".ErrorDetail_ES := 'Fallo de objeto tecnologico husillo - presionar Ack/Reset para borrar';
	        IF #State <> #STATE_ERROR AND #State <> 0 AND #State <> #STATE_PRE_SCAN THEN
	            #State := #STATE_ERROR;
	        END_IF;
	    END_IF;
	    #prevTOFaultSpindle := TRUE;
	ELSE
	    #prevTOFaultSpindle := FALSE;
	END_IF;

	// Limit monitor
	#fbLimitMonitor(ActualPos_X := #Axis_X.ActualPosition,
	                ActualPos_Z := #Axis_Z.ActualPosition,
	                Homed_X := #Axis_X.StatusBits.HomingDone,
	                Homed_Z := #Axis_Z.StatusBits.HomingDone,
	                HW_NC_X_Min := #HW_NC_X_Min,
	                HW_NC_X_Max := #HW_NC_X_Max,
	                HW_NC_Z_Min := #HW_NC_Z_Min,
	                HW_NC_Z_Max := #HW_NC_Z_Max,
	                HW_PNP_X_Min := #HW_PNP_X_Min,
	                HW_PNP_X_Max := #HW_PNP_X_Max,
	                HW_PNP_Z_Min := #HW_PNP_Z_Min,
	                HW_PNP_Z_Max := #HW_PNP_Z_Max);
	// NOTE: FB_LimitMonitor itself now checks soft limits only for HOMED axes
	// (Homed_X/Z inputs = StatusBits.HomingDone) -- an un-homed axis can never trip a
	// soft limit. The state bypasses below remain as defense in depth:
	// During homing the axis may move outside soft limits (moving toward home switch).
	// All four homing-related states are bypassed: PRE_HOME_CLR, HOMING, POST_HOME_CLR,
	// and STOP_GOHOME. Without bypassing PRE/POST_HOME_CLR the clearance moves could
	// trip a spurious soft-limit fault before homing even begins (TO position = 0 after restart).
	// STATE_MANUAL and STATE_PNP_HALT are also bypassed: manual mode enforces soft limits
	// via directional jog gating + MoveAbsolute target rejection (never faults, so the
	// operator can always jog back into range).
	// STATE_PRE_SCAN(12) and STATE_STARTING(10) are bypassed because:
	//   PRE_SCAN: pure software validation, no motion -- TO position may be stale from last run.
	//   STARTING: contactors just closing, drives not yet ready -- homing will establish real position.
	// HW limit switch faults are caught by TO â†’ MC_Home.Error â†’ handled in state machine.
	IF #State = #STATE_HOMING OR #State = #STATE_STOP_GOHOME
	    OR #State = #STATE_PRE_HOME_CLR OR #State = #STATE_POST_HOME_CLR
	    OR #State = #STATE_MANUAL OR #State = #STATE_PNP_HALT
	    OR #State = #STATE_PRE_SCAN OR #State = #STATE_STARTING THEN
	    #SafeToRun := #fbSafetyMonitor.SafeToRun;   // Soft limit bypass
	ELSE
	    #SafeToRun := #fbSafetyMonitor.SafeToRun AND NOT #fbLimitMonitor.LimitError;
	END_IF;

	// Safety error handling
	// NOTE: Alarm is only raised from active states such as RUNNING/MANUAL.
	// No new alarm is raised in STOPPED (0) or ERROR (999) state;
	// this prevents drive enable delay after ACK/Reset from creating spurious alarms.
	IF NOT #fbSafetyMonitor.SafeToRun AND #fbSafetyMonitor.ErrorCode <> 0 THEN
	    IF NOT #prevSafetyError AND #State <> 0 AND #State <> #STATE_ERROR THEN
	        #newErrorFlag := TRUE;
	        #newErrorCode := #fbSafetyMonitor.ErrorCode;
	    END_IF;
	    IF #State <> 0 AND #State <> #STATE_ERROR THEN
	        #State := #STATE_ERROR;
	    END_IF;
	    #prevSafetyError := TRUE;
	ELSE
	    #prevSafetyError := FALSE;
	END_IF;

	// Soft limit error handling -- triggers STATE_ERROR when axis exceeds configured soft limits.
	// Un-homed axes never trip (FB_LimitMonitor Homed_X/Z gating -- position is meaningless
	// before the reference seek completes).
	// NC hardware limit switches are removed from LimitMonitor; TO handles them natively.
	// Bypassed in all four homing-related states: during homing the axis may legitimately
	// travel outside the configured limits while seeking the reference switch.
	// STATE_MANUAL and STATE_PNP_HALT also bypassed: manual mode enforces soft limits via
	// directional jog gating + MoveAbsolute target rejection instead of faulting.
	// STATE_PRE_SCAN(12) and STATE_STARTING(10) bypassed: TO position may be stale
	// from the previous run; firing here would abort startup for a position that was valid last run.
	IF #fbLimitMonitor.LimitError AND #fbLimitMonitor.ErrorCode <> 0
	    AND #State <> #STATE_HOMING AND #State <> #STATE_STOP_GOHOME
	    AND #State <> #STATE_PRE_HOME_CLR AND #State <> #STATE_POST_HOME_CLR
	    AND #State <> #STATE_MANUAL AND #State <> #STATE_PNP_HALT
	    AND #State <> #STATE_PRE_SCAN AND #State <> #STATE_STARTING
	    AND #State <> #STATE_STOPPED AND #State <> #STATE_ERROR THEN
	    #newErrorFlag := TRUE;
	    #newErrorCode := #fbLimitMonitor.ErrorCode;
	    #State := #STATE_ERROR;
	END_IF;

